Yaskawa INFORM job: SKRZYNIA_4840_0_STOPNI_2OBR.JBI

/JOB
//NAME SKRZYNIA_4840_0_STOPNI_2OBR
///FOLDERNAME 02-SKRZYNIE_JOBS
//POS
///NPOS 694,694,0,51,0,0
///TOOL 0
///POSTYPE PULSE
///PULSE
C00000=1055,-24125,84372,288,19725,204
C00001=0,-15438,65714,0,-68532,0
C00002=4718,-16587,59952,3396,-65485,-935
C00003=32997,-21499,42555,27623,-61436,21376
C00004=31759,-20688,42932,26837,-60850,21559
C00005=28987,-21156,42712,24818,-60442,22222
C00006=33447,-21964,42352,27886,-61721,21330
C00007=37687,-23357,41794,30651,-63289,20620
C00008=38979,-19018,48057,32961,-64962,20678
C00009=37261,-18075,48526,31902,-64209,20901
C00010=35830,-17198,48994,31015,-63571,21092
C00011=34080,-17614,48768,29780,-63290,21485
C00012=37261,-18075,48526,31902,-64209,20901
C00013=4718,-16587,59952,3396,-65485,-935
C00014=32997,-21499,42555,27623,-61436,21376
C00015=31759,-20688,42932,26837,-60850,21559
C00016=28987,-21156,42712,24818,-60442,22222
C00017=33447,-21964,42352,27886,-61721,21330
C00018=37687,-23357,41794,30651,-63289,20620
C00019=38979,-19018,48057,32961,-64962,20678
C00020=37261,-18075,48526,31902,-64209,20901
C00021=35830,-17198,48994,31015,-63571,21092
C00022=34080,-17614,48768,29780,-63290,21485
C00023=37261,-18075,48526,31902,-64209,20901
C00024=47373,-21912,40596,41149,-66086,26950
C00025=45033,-20851,41104,39798,-65001,27223
C00026=42790,-19693,41704,38494,-63946,27495
C00027=41070,-20182,41442,37324,-63566,27891
C00028=45033,-20851,41104,39798,-65001,27223
C00029=45033,-20851,41104,39798,-65001,27223
C00030=59624,-29540,14278,64846,-60867,16042
C00031=57357,-28542,14780,63940,-59509,16120
C00032=56188,-29140,14476,63237,-58995,16387
C00033=59588,-29370,14363,64862,-60819,16012
C00034=54896,-47461,-5979,49852,-59285,4360
C00035=10104,-46603,4759,11228,-37390,-5046
C00036=0,-52280,40443,0,6876,0
C00037=1529,-42140,58025,-5964,2417,3265
C00038=0,-38374,23626,-1605,-51738,268
C00039=63773,-21017,30186,64198,-68685,10387
C00040=61397,-24232,22270,64115,-66256,9272
C00041=59945,-23569,22659,63511,-65413,9334
C00042=58737,-24250,22260,62835,-64893,9588
C00043=61397,-24232,22270,64115,-66256,9272
C00044=45044,-23015,37260,35797,-71879,25522
C00045=39973,-29571,18873,35060,-63052,24165
C00046=38620,-28701,19269,34339,-62304,24363
C00047=36409,-29254,19014,32896,-61805,24958
C00048=44451,-29039,21934,37281,-65892,23702
C00049=49472,-39353,6917,53118,-50908,20251
C00050=45058,-39356,3832,51653,-47640,20099
C00051=42883,-38319,4163,50577,-46309,20295
C00052=40255,-38926,3967,48502,-45334,21060
C00053=46774,-39679,3737,52663,-48537,19827
C00054=48708,-40455,3517,53615,-49689,19657
C00055=43798,-39237,3871,50850,-47027,20335
C00056=41951,-38324,4161,49930,-45891,20507
C00057=39836,-38844,3994,48234,-45126,21137
C00058=48489,-40338,3551,53521,-49551,19665
C00059=1148,-56354,34370,-23,3827,-9
C00060=1148,-56354,34370,-23,3827,-9
C00061=48489,-40338,3551,53521,-49551,19665
C00062=44432,-39026,3936,51363,-47247,20139
C00063=42487,-38069,4248,50403,-46050,20315
C00064=39061,-38795,4009,47695,-44769,21310
C00065=44432,-39026,3936,51363,-47247,20139
C00066=43521,-36748,12770,50182,-45701,23408
C00067=41846,-35383,13175,49516,-44517,23399
C00068=39971,-34448,13485,48491,-43408,23582
C00069=37453,-34980,13306,46330,-42542,24334
C00070=41846,-35383,13175,49516,-44517,23399
C00071=78369,-41260,16071,67181,-65880,21417
C00072=137,-45861,52341,97,-67596,-14
C00073=-31499,-58302,-23356,15027,12889,-13082
C00074=-52768,-43016,-26078,18373,38595,-18774
C00075=-89470,-32103,-32973,29905,69139,-31512
C00076=-68838,-26884,-24872,16972,64732,-23076
C00077=-53036,-11528,-12218,12363,64665,-17409
C00078=-51536,-9474,-10276,11905,64649,-16876
C00079=-51739,-9114,-7787,12104,63269,-17104
C00080=-53036,-11528,-12218,12363,64665,-17409
C00081=-17541,-26226,-24397,927,59032,-5038
C00082=-17541,-26226,-24397,927,59032,-5038
C00083=-16950,-23991,-22741,715,59568,-4818
C00084=-17036,-23563,-20101,755,58071,-4857
C00085=-17541,-26226,-24397,927,59032,-5038
C00086=34102,-23192,-21614,-15638,64271,13209
C00087=33423,-21885,-20599,-15423,64418,12942
C00088=32426,-19856,-18975,-15106,64629,12551
C00089=32578,-19611,-17013,-15290,63535,12762
C00090=33423,-21885,-20599,-15423,64418,12942
C00091=59339,-6070,-6417,-20979,72191,20891
C00092=59339,-6070,-6417,-20979,72191,20891
C00093=57897,-4256,-4562,-20702,71913,20431
C00094=58108,-3992,-2506,-20878,70835,20713
C00095=59339,-6070,-6417,-20979,72191,20891
C00096=42744,-35904,-30225,-18322,62562,16651
C00097=-53036,-11528,-12218,12363,64665,-17409
C00098=-77982,-26538,-29134,27151,66629,-27745
C00099=-70983,-8594,-1966,26503,59809,-49670
C00100=-80152,19776,40785,37351,72704,-50428
C00101=-79984,20154,42529,37516,71911,-50638
C00102=-79233,18397,40079,37458,71885,-50340
C00103=-79984,20154,42529,37516,71911,-50638
C00104=-73519,23289,38838,28890,77081,-45618
C00105=-73519,24511,42682,29072,75582,-46027
C00106=-73519,23289,38838,28890,77081,-45618
C00107=-88897,15706,42282,50101,71325,-56974
C00108=-88897,15706,42282,50101,71325,-56974
C00109=-87612,12343,37838,50071,70996,-56519
C00110=-85283,14202,40272,50301,69633,-56165
C00111=-87338,12550,38107,50098,70839,-56476
C00112=-84952,-1789,13569,34660,47724,-58955
C00113=-67641,-1674,11109,10330,44856,-44725
C00114=-66443,961,13975,9688,44721,-44210
C00115=-67641,-1674,11109,10330,44856,-44725
C00116=-67641,-376,15347,10694,42950,-44967
C00117=-67641,-1674,11109,10330,44856,-44725
C00118=-79040,417,20398,15965,28992,-57786
C00119=-76655,5212,30978,15501,25024,-57306
C00120=-76655,6949,35816,16758,23084,-57955
C00121=-76655,5212,30978,15501,25024,-57306
C00122=-74761,6919,33010,13466,24593,-56049
C00123=-80460,-2874,12270,15804,32253,-57809
C00124=-61258,-29124,-13156,26560,43617,-22150
C00125=-30420,-40507,-29240,27153,53235,15188
C00126=-18589,-38725,-21450,23338,47896,18931
C00127=-17722,-35233,-16455,23322,46926,19051
C00128=-17722,-33749,-12435,23948,45421,18620
C00129=-17722,-33892,-12819,23887,45564,18661
C00130=-16677,-31133,-11209,23138,46167,19311
C00131=-17819,-35820,-17540,23246,47228,19090
C00132=-74104,-11494,-6266,31916,75042,4269
C00133=-71226,-7329,2631,32115,71468,4273
C00134=-71226,-6504,5446,32343,70365,3922
C00135=-71226,-6611,5086,32313,70505,3967
C00136=-68386,-4058,7675,32040,69573,4789
C00137=-73314,-9412,-353,32206,72648,3829
C00138=51751,-31069,-22965,-10739,49070,48663
C00139=49028,-23852,-11575,-9841,46366,47823
C00140=49028,-23004,-8935,-10039,45204,47956
C00141=49028,-23118,-9286,-10013,45357,47939
C00142=47000,-20813,-7527,-8928,45644,47024
C00143=50476,-26208,-15307,-10408,47325,48332
C00144=90602,-5375,6902,-38786,69848,59444
C00145=83174,19950,50269,-44999,67580,58220
C00146=82362,17902,47383,-44926,67511,57879
C00147=83515,19072,48341,-44798,68200,58056
C00148=78091,19382,40247,-36371,72286,52960
C00149=78091,20664,44011,-36670,70997,53443
C00150=78091,19382,40247,-36371,72286,52960
C00151=88699,7296,38566,-55615,63182,60372
C00152=86803,3068,32674,-55410,62638,59657
C00153=84852,4315,34115,-55564,61561,59330
C00154=86803,3068,32674,-55410,62638,59657
C00155=92770,-2803,21719,-53893,67577,59421
C00156=73393,-10627,10934,-27897,30744,62458
C00157=70789,-6606,18800,-27824,27830,62140
C00158=69654,-4593,20814,-26755,27596,61444
C00159=70789,-6606,18800,-27824,27830,62140
C00160=70789,-5070,23059,-29482,26284,63017
C00161=70789,-6606,18800,-27824,27830,62140
C00162=83486,-8736,6503,-27040,35338,66550
C00163=77831,-2041,26192,-25270,18452,68895
C00164=77967,1961,32070,-26860,17569,69698
C00165=77967,5243,40752,-32914,14549,72656
C00166=77967,1961,32070,-26860,17569,69698
C00167=74560,4730,35257,-21622,16551,66717
C00168=77967,1961,32070,-26860,17569,69698
C00169=81109,-22356,2664,-22493,33121,60116
C00170=86168,-49730,-13668,-23926,46819,49343
C00171=44183,-52048,-7537,-24795,46064,51426
C00172=0,-52280,40443,0,6876,0
C00173=0,-52280,40443,0,6876,0
C00174=33629,-57276,-6399,46271,-24969,-2804
C00175=75493,-63502,-64712,103874,-64610,-6298
C00176=47968,-58405,-62693,109749,-46222,-10681
C00177=44214,-60060,-65896,114303,-43519,-9276
C00178=55379,-67378,-68041,108237,-48773,-4935
C00179=62671,-64213,-64640,104431,-56093,-7372
C00180=28458,-50318,6850,47420,-25887,-3347
C00181=0,-52280,40443,0,6876,0
C00182=1055,-24125,84372,288,19725,204
C00183=0,-15438,65714,0,-68532,0
C00184=0,-15438,65714,966,-70097,42926
C00185=69988,-9219,57065,61610,-82752,27767
C00186=63113,-6157,59685,58080,-79692,28271
C00187=46135,-5501,68028,40160,-75108,29748
C00188=49471,-5188,67710,43421,-76082,29577
C00189=63113,-6157,59685,58080,-79692,28271
C00190=69988,-9219,57065,61610,-82752,27767
C00191=0,-15438,65714,966,-70097,42926
C00192=0,-15438,65714,0,-68532,0
C00193=1055,-24125,84372,288,19725,204
C00194=1055,-24125,84372,288,19725,204
C00195=0,-41971,13909,0,6774,1
C00196=-55064,-17017,13106,20113,45767,-35735
C00197=-85641,-3161,12660,31281,67420,-55579
C00198=-77611,9747,38455,32702,57795,-55547
C00199=-77611,9747,38455,32702,57795,-55547
C00200=-80481,23547,61641,37204,60115,-56891
C00201=-80479,11681,28780,33754,71138,-52780
C00202=-73572,15026,34389,33675,67405,-51294
C00203=-73572,20195,49236,35290,62248,-53161
C00204=-82806,26311,53816,38180,73291,-53604
C00205=-71695,3747,16001,30713,64750,-51022
C00206=-70421,5575,20105,30867,63066,-51036
C00207=-35543,-20105,-5144,22821,50284,-40173
C00208=-37830,-23193,-8618,23571,50957,-40982
C00209=11136,-28839,-12562,1025,41780,-20887
C00210=20486,-27077,-7346,-12554,38415,-10736
C00211=59545,-9921,5571,-27063,51925,3267
C00212=55110,-17412,-5825,-19778,50988,-2825
C00213=79390,11759,28162,-35512,71262,52960
C00214=74811,13878,33986,-35807,67493,52464
C00215=74942,18762,48004,-37392,62815,54352
C00216=76815,18630,46530,-37158,64288,54543
C00217=79390,11759,28162,-35512,71262,52960
C00218=10831,-54278,-29128,-6468,39852,-5090
C00219=-67200,-10549,24402,-3189,24913,-39001
C00220=-75122,-2194,12822,3152,39225,-43427
C00221=-77516,10189,32861,8493,33365,-45533
C00222=-75154,17575,49272,7885,27457,-44928
C00223=-68113,9932,38901,1157,28472,-40453
C00224=-67114,5383,31515,9208,32648,-43213
C00225=-66450,3998,29285,10896,33890,-43630
C00226=-66374,3101,28136,14657,35566,-44954
C00227=-66576,452,24763,27028,43375,-49112
C00228=-69928,4230,30673,35488,50431,-52676
C00229=-77050,-3138,8526,33226,61087,-51698
C00230=-67200,-10549,24402,-3189,24913,-39001
C00231=0,-52280,40443,83103,28146,-16510
C00232=99993,-20782,22705,-13349,24734,56519
C00233=67200,-10549,24402,3189,24913,39001
C00234=75122,-2194,12822,-3152,39225,43427
C00235=74323,5203,27259,-5972,33194,43789
C00236=74015,16414,48063,-6821,27325,44224
C00237=56519,1138,28747,9235,29393,33453
C00238=55467,619,28251,10155,29461,32830
C00239=56374,-724,25854,4078,30541,35419
C00240=56480,-7201,15910,-17697,38451,43334
C00241=68252,956,25699,-34035,49810,51639
C00242=77050,-3138,8526,-33226,61087,51698
C00243=67200,-10549,24402,3189,24913,39001
C00244=0,-52280,40443,-83103,28146,16510
C00245=-99993,-20782,22705,13349,24734,-56519
C00246=-91125,453,39555,30378,52425,-51131
C00247=-81425,-5449,14825,37552,56592,-47667
C00248=-81425,-10835,-2515,34915,62871,-45127
C00249=-79239,4305,16082,37593,68846,-50182
C00250=-81302,5892,27588,46359,62943,-54679
C00251=-82227,19402,59913,51524,57300,-60581
C00252=-84844,8890,27031,38640,69740,-53449
C00253=-90096,4679,14083,37467,76581,-51973
C00254=-87885,29238,52923,40761,81198,69685
C00255=-84355,23847,39024,40698,83720,72224
C00256=-81960,27335,46957,41070,80536,71891
C00257=-82643,24718,50492,48951,72637,70260
C00258=-90480,18737,31939,47254,81986,71631
C00259=-94217,10634,17426,46901,86469,-59967
C00260=-81425,-10835,-2515,34915,62871,-45127
C00261=-81425,-5449,14825,37552,56592,-47667
C00262=-94290,-610,44819,32366,49686,-53459
C00263=0,-55136,17047,60468,32096,-4233
C00264=99993,-20782,22705,-13349,24734,56519
C00265=91125,453,39555,-30378,52425,51131
C00266=81425,-5449,14825,-37552,56592,47667
C00267=81425,-10835,-2515,-34915,62871,45127
C00268=79239,4305,16082,-37593,68846,50182
C00269=83239,4964,30263,-50637,62037,57149
C00270=83991,16425,61235,-57769,55250,63273
C00271=93928,7973,40920,-53095,64494,61640
C00272=75109,22299,39152,-26915,78743,47998
C00273=79256,17348,34699,-33448,76412,88212
C00274=79932,23608,50901,-39863,71219,88955
C00275=76220,30771,63034,-41386,67395,88927
C00276=86322,16060,37848,-39554,76452,89287
C00277=87424,-1569,9538,-38190,72401,52253
C00278=81425,-10835,-2515,-34915,62871,45127
C00279=92850,-11266,9233,-39092,60986,50964
C00280=28366,-40369,19479,-5635,23506,17663
C00281=-80334,-19501,31260,21216,42469,-40219
C00282=-80621,-32280,-9061,25825,59412,-41877
C00283=-80621,-37319,-22868,24573,64555,-40576
C00284=-75108,-2453,16462,35304,60348,-42510
C00285=-72231,7240,33473,36511,55681,-43130
C00286=-35770,-19109,7486,28512,40799,-31761
C00287=-39606,-22901,-1163,28356,44724,-32188
C00288=15344,-29112,-5358,-2858,33820,-6852
C00289=13390,-24012,2637,-1527,32105,-7853
C00290=57983,-8601,15571,-27088,42703,12849
C00291=60973,-17187,4937,-27817,44388,13718
C00292=60973,-17187,4937,-27817,44388,13718
C00293=-13287,-42463,-12044,19170,31021,-23010
C00294=-17374,-21287,20534,22794,29118,-26096
C00295=13276,-20759,18622,-1911,29377,-7028
C00296=39924,-14247,19329,-14795,35999,4396
C00297=41528,-14133,18797,-15449,36702,5040
C00298=57001,-5890,26499,-21893,40771,11494
C00299=64054,-19541,3059,-29141,44956,15011
C00300=51466,-33957,-1499,-46586,51805,23434
C00301=17032,-20770,22044,-28854,30468,11088
C00302=-9868,-18638,14971,-8492,38486,-5199
C00303=-40562,-13194,19800,9508,35447,-20184
C00304=-41848,-12620,20103,10165,35810,-20773
C00305=-57278,-4046,28217,17578,39066,-27653
C00306=-71680,-19835,10874,33863,39440,-36917
C00307=-20806,-37586,-12792,9951,42782,-18031
C00308=29087,-45372,27330,-13325,19529,9021
C00309=0,-52280,40443,0,6876,0
C00310=0,-52280,40443,0,6876,0
C00311=0,-52280,40443,0,6876,0
C00312=0,-52280,40443,0,-40718,0
C00313=32359,-35955,27464,28918,-49457,29587
C00314=33244,-30989,28192,31082,-46894,28340
C00315=21151,-27492,32720,20239,-44670,31873
C00316=21536,-57229,-33277,36819,-24396,22621
C00317=20406,-52755,-25486,23563,-35235,28276
C00318=29904,-46498,-2819,27004,-47536,28031
C00319=45803,-31685,22885,64496,-39050,18987
C00320=0,-52277,40442,0,6872,2
C00321=0,-38538,66749,0,-898,0
C00322=0,-52280,40443,0,-79033,35417
C00323=46775,-35113,22190,42926,-67531,20697
C00324=52587,-26056,25345,47610,-66542,17970
C00325=45775,-25572,24450,44032,-63158,18875
C00326=45891,-27794,19511,44698,-62000,18216
C00327=53914,-29436,22058,48262,-67266,17843
C00328=63113,-6157,59685,58080,-79692,28271
C00329=47789,-6280,67353,41142,-75661,29541
C00330=47201,-5612,67930,40804,-75418,29594
C00331=49592,-5172,67757,43430,-76113,29541
C00332=58547,-7653,65645,48613,-79176,28479
C00333=46775,-35113,22190,42926,-67531,20697
C00334=0,-52280,40443,0,-79033,35417
C00335=0,-38922,70509,0,-71891,28081
C00336=0,-38922,70509,0,-71891,28081
C00337=36958,-10079,72709,30464,-66560,20948
C00338=30513,-4130,80544,25739,-66271,22156
C00339=4090,-36983,1084,-1138,-53633,29170
C00340=13946,-45192,10090,9828,-39459,25958
C00341=404,-42897,57020,-1574,2523,869
C00342=0,-52280,40443,0,6876,0
C00343=-99253,-13690,44082,59847,13407,-31313
C00344=-87814,-12734,20141,45739,-14352,-64418
C00345=-86669,-6582,30812,41148,-16781,-62025
C00346=-85055,-5827,31548,44003,-17420,-63187
C00347=-85971,-6262,31124,42409,-17052,-62539
C00348=-86650,-5303,32069,41395,-16716,-62141
C00349=-94954,-14494,-1860,-7818,15857,-59130
C00350=-94509,1544,30797,-849,15127,-60471
C00351=-94509,4151,37772,-1041,12286,-60378
C00352=-88011,-10036,27574,37950,-16527,-60658
C00353=-86125,-12470,22545,29004,-25567,-58412
C00354=-85732,-21202,11427,30682,-24763,-59235
C00355=-84150,-10929,23786,31981,-25941,-59678
C00356=-83036,-10419,24246,33504,-26268,-60308
C00357=-84150,-10929,23786,31981,-25941,-59678
C00358=-85291,-9507,25078,30650,-25411,-59154
C00359=-84150,-10929,23786,31981,-25941,-59678
C00360=-85786,-16909,14677,31743,-23900,-59790
C00361=-84150,-10498,24888,31517,-26306,-59436
C00362=-83174,-10052,25293,32841,-26587,-59984
C00363=-84150,-10498,24888,31517,-26306,-59436
C00364=-85258,-9112,26156,30226,-25800,-58928
C00365=-84150,-10498,24888,31517,-26306,-59436
C00366=-87841,-18519,13420,28367,-23534,-58339
C00367=-84150,-10465,24972,31484,-26336,-59417
C00368=-83241,-10052,25348,32714,-26598,-59924
C00369=-84150,-10465,24972,31484,-26336,-59417
C00370=-85145,-9228,26102,30329,-25881,-58963
C00371=-84150,-10465,24972,31484,-26336,-59417
C00372=-86371,-18277,13606,30568,-23951,-59265
C00373=-84345,-11688,21985,32461,-25312,-59957
C00374=-83211,-11173,22442,34044,-25650,-60618
C00375=-84345,-11688,21985,32461,-25312,-59957
C00376=-85283,-10526,23025,31366,-24861,-59525
C00377=-84345,-11688,21985,32461,-25312,-59957
C00378=-86191,-19647,12567,30467,-24278,-59187
C00379=-84345,-10877,24073,31552,-26006,-59481
C00380=-83051,-10286,24607,33321,-26381,-60213
C00381=-84345,-10877,24073,31552,-26006,-59481
C00382=-85179,-9842,25009,30582,-25619,-59100
C00383=-84345,-10877,24073,31552,-26006,-59481
C00384=-85438,-18022,14839,31140,-24818,-59429
C00385=-84247,-11820,22550,32049,-25753,-59727
C00386=-84104,-10976,23642,32111,-25899,-59738
C00387=-82990,-10465,24105,33639,-26227,-60372
C00388=-84104,-10976,23642,32111,-25899,-59738
C00389=-84898,-9998,24525,31196,-25529,-59378
C00390=-84104,-10976,23642,32111,-25899,-59738
C00391=-86610,-16845,14732,30573,-23614,-59301
C00392=-84104,-10864,23927,31990,-25993,-59674
C00393=-82824,-10273,24459,33737,-26370,-60397
C00394=-84104,-10864,23927,31990,-25993,-59674
C00395=-84789,-10021,24690,31200,-25673,-59363
C00396=-84104,-10864,23927,31990,-25993,-59674
C00397=-83806,-19585,12613,33764,-25080,-60559
C00398=-83924,-10205,25475,31619,-26533,-59453
C00399=-82780,-9675,25960,33156,-26866,-60087
C00400=-83924,-10205,25475,31619,-26533,-59453
C00401=-84478,-9530,26093,30986,-26280,-59206
C00402=-83924,-10205,25475,31619,-26533,-59453
C00403=-87149,-17993,13826,29513,-23647,-58830
C00404=-84920,-13182,20975,31162,-25481,-59361
C00405=-83711,-10572,24852,32056,-26475,-59649
C00406=-82779,-10142,25241,33309,-26748,-60166
C00407=-83711,-10572,24852,32056,-26475,-59649
C00408=-84370,-9774,25579,31305,-26170,-59356
C00409=-83711,-10572,24852,32056,-26475,-59649
C00410=-83642,-3679,42021,23358,-36761,-56118
C00411=-85886,-5975,41264,18964,-40261,-54782
C00412=-83919,-11632,22322,32811,-25616,-60079
C00413=-82884,-11162,22742,34234,-25925,-60671
C00414=-83919,-11632,22322,32811,-25616,-60079
C00415=-84723,-10654,23196,31887,-25230,-59715
C00416=-83919,-11632,22322,32811,-25616,-60079
C00417=-87348,-16035,7353,17528,-35245,-56477
C00418=-86244,-15062,8172,18754,-35315,-57058
C00419=-86244,-16649,3638,19674,-33501,-57585
C00420=-85308,-16228,3988,20718,-33648,-58082
C00421=-86244,-16649,3638,19674,-33501,-57585
C00422=-86740,-15973,4201,19194,-33277,-57362
C00423=-86244,-16649,3638,19674,-33501,-57585
C00424=-73780,-8639,20128,34258,-51705,-52097
C00425=-90711,-17528,-28778,11328,-28245,-57111
C00426=-92565,-19610,-33223,7138,-24591,-57051
C00427=-91512,-19116,-32812,8551,-24603,-57834
C00428=-92565,-19610,-33223,7138,-24591,-57051
C00429=-93003,-18716,-32476,6600,-24397,-56752
C00430=-92565,-19610,-33223,7138,-24591,-57051
C00431=-92565,-19610,-33223,7138,-24591,-57051
C00432=-95836,-54375,-51122,6031,-17685,-48210
C00433=-95836,-54375,-51122,6031,-17685,-48210
C00434=-43821,-47238,-2775,-3022,56549,-3681
C00435=-20126,-26882,59542,2406,16879,-9162
C00436=-20126,-26882,59542,2406,16879,-9162
C00437=98601,-10520,92678,4674,-40855,-9615
C00438=95537,-19831,-2695,-2933,-44471,35837
C00439=92548,-20391,-28429,-6186,-30623,55200
C00440=91429,-17018,-28974,-8057,-27827,56250
C00441=91429,-17018,-28974,-8057,-27827,56250
C00442=90371,-16495,-28521,-9286,-27856,56953
C00443=91429,-17018,-28974,-8057,-27827,56250
C00444=92033,-15799,-27911,-7415,-27588,55880
C00445=91429,-17018,-28974,-8057,-27827,56250
C00446=92548,-20391,-28429,-6186,-30623,55200
C00447=91156,-15018,-4648,-8036,-38181,54813
C00448=90585,-14766,-4428,-8565,-38201,55100
C00449=88830,-13959,-3717,-10186,-38284,55977
C00450=89897,-14456,-4157,-9202,-38230,55445
C00451=90761,-12944,-2809,-8452,-37927,55043
C00452=89897,-14456,-4157,-9202,-38230,55445
C00453=89670,-8466,73559,-9449,-60959,55261
C00454=89910,-11217,67535,-9455,-58896,55399
C00455=85786,-16735,14816,-31782,-23869,59812
C00456=83514,-12996,17929,-35760,-24132,61552
C00457=82251,-12406,18443,-37550,-24551,62308
C00458=83514,-12996,17929,-35760,-24132,61552
C00459=84258,-12095,18717,-34917,-23742,61217
C00460=83514,-12996,17929,-35760,-24132,61552
C00461=87149,-17993,13826,-29513,-23647,58830
C00462=83118,-12818,18089,-36330,-24263,61791
C00463=81915,-12248,18589,-38020,-24666,62504
C00464=83118,-12818,18089,-36330,-24263,61791
C00465=83897,-11882,18912,-35460,-23856,61445
C00466=83118,-12818,18089,-36330,-24263,61791
C00467=83806,-19585,12613,-33764,-25080,60559
C00468=82998,-13006,17925,-36445,-24332,61826
C00469=81675,-12378,18472,-38297,-24777,62607
C00470=82998,-13006,17925,-36445,-24332,61826
C00471=83876,-11958,18841,-35466,-23874,61442
C00472=82998,-13006,17925,-36445,-24332,61826
C00473=86610,-16845,14732,-30573,-23614,59301
C00474=82493,-13239,17725,-37070,-24559,62089
C00475=81406,-12724,18174,-38578,-24928,62723
C00476=82493,-13239,17725,-37070,-24559,62089
C00477=83436,-12134,18690,-36041,-24064,61684
C00478=82493,-13239,17725,-37070,-24559,62089
C00479=84814,-16043,15376,-33312,-24093,60464
C00480=82555,-13613,17404,-36910,-24580,62015
C00481=81384,-13062,17878,-38534,-24974,62698
C00482=82555,-13613,17404,-36910,-24580,62015
C00483=83566,-12434,18427,-35805,-24047,61580
C00484=82555,-13613,17404,-36910,-24580,62015
C00485=86191,-19647,12567,-30467,-24278,59187
C00486=82500,-13648,17375,-36975,-24607,62039
C00487=81467,-13161,17792,-38413,-24955,62645
C00488=82500,-13648,17375,-36975,-24607,62039
C00489=83481,-12505,18364,-35905,-24087,61617
C00490=82500,-13648,17375,-36975,-24607,62039
C00491=86371,-18277,13606,-30568,-23951,59265
C00492=82904,-13790,17251,-36416,-24470,61808
C00493=81715,-13237,17726,-38081,-24865,62509
C00494=82904,-13790,17251,-36416,-24470,61808
C00495=83686,-12878,18037,-35556,-24055,61469
C00496=82904,-13790,17251,-36416,-24470,61808
C00497=87841,-18519,13420,-28367,-23534,58339
C00498=82748,-13879,17174,-36603,-24542,61883
C00499=81692,-13388,17594,-38077,-24893,62505
C00500=82748,-13879,17174,-36603,-24542,61883
C00501=83607,-12881,18032,-35663,-24082,61515
C00502=82748,-13879,17174,-36603,-24542,61883
C00503=85786,-16909,14677,-31743,-23900,59790
C00504=82520,-14198,16902,-36833,-24674,61972
C00505=81460,-13708,17319,-38301,-25026,62591
C00506=82520,-14198,16902,-36833,-24674,61972
C00507=83571,-12989,17938,-35691,-24113,61524
C00508=82520,-14198,16902,-36833,-24674,61972
C00509=85732,-21202,11427,-30682,-24763,59235
C00510=82398,-14365,16763,-36952,-24745,62014
C00511=81172,-13798,17245,-38643,-25153,62725
C00512=82398,-14365,16763,-36952,-24745,62014
C00513=83600,-12984,17944,-35650,-24102,61504
C00514=82398,-14365,16763,-36952,-24745,62014
C00515=86140,-12802,12665,-93523,-10743,85795
C00516=86140,-12802,12665,-93523,-10743,85795
C00517=85030,-12289,13120,-93723,-11463,85776
C00518=86140,-12802,12665,-93523,-10743,85795
C00519=86958,-11660,13681,-94506,-10238,86349
C00520=85239,-16743,-4327,42764,21357,45785
C00521=86674,107,23869,25042,24033,51593
C00522=86674,2327,30134,27824,21680,50173
C00523=87715,-15254,10554,-91589,-9692,85040
C00524=85045,-36869,-4353,-28502,-22832,52282
C00525=0,-24029,84339,0,19981,0
C00526=0,-24029,84339,0,19981,0
C00527=3172,-24246,80980,3465,15913,689
C00528=-86563,-26985,13879,10257,-21548,-45530
C00529=-86191,-19647,12567,30467,-24278,-59187
C00530=-83221,-13587,17636,37793,-25116,-62228
C00531=-91978,-13833,14560,12391,-18633,-51524
C00532=-94992,-13830,14285,1276,-18012,-46664
C00533=-84074,-17488,11256,38660,-23649,-62784
C00534=-73679,-33270,1000,44272,-31600,-64253
C00535=-86926,-60758,23267,6576,1160,-9545
C00536=0,-52280,40443,0,6876,0
C00537=82475,-58079,26734,835,4084,4444
C00538=97932,-26840,7691,8784,-23444,42538
C00539=87166,-16607,16322,-25365,-24201,56345
C00540=84699,-11354,21752,-29145,-24735,57949
C00541=84804,-11023,22730,-28561,-25071,57659
C00542=85100,-26994,10417,-24982,-28140,55821
C00543=0,-52280,40443,0,6876,0
C00544=0,-52280,40443,0,6876,0
C00545=-90140,-60305,18108,-2708,1721,-7625
C00546=-95594,-27428,6866,-4663,-19832,-42154
C00547=-98688,-13767,16447,-18366,-10080,-35766
C00548=-98967,-3050,34440,-28957,-8622,-29685
C00549=-100063,5316,51567,-32262,-10006,-27560
C00550=-94586,18541,64268,-6451,10518,-43578
C00551=-95535,2380,25473,239,27557,-47214
C00552=-91259,3120,34463,-5130,22041,-43946
C00553=-95333,12702,45733,36,21375,-47085
C00554=-99268,-13088,27343,-18620,-14105,-35021
///LIMIT ON
C00555=-90140,-60305,18108,-2708,1721,-7625
///LIMIT OFF
C00556=0,-52280,40443,0,6876,0
C00557=84259,-57935,27522,-3761,3673,6310
C00558=86507,-39672,4297,-27618,-16640,46340
C00559=73669,-37119,-20783,-92053,-19719,85232
C00560=86539,-20830,1725,-71850,-11773,76853
C00561=90325,-18913,6238,-62161,-7452,70888
C00562=97679,-11879,12650,-55334,4229,66281
C00563=98389,-8856,11720,-15676,14634,48538
C00564=96255,-748,20886,-3277,24061,38276
C00565=95132,-6008,10010,1655,28777,36730
C00566=94050,-4188,7205,-2481,41508,36662
C00567=98126,4908,16834,-5042,41918,38535
C00568=100487,-9453,-1206,-10413,41328,41147
C00569=96250,-19428,-8283,-4838,27297,37910
C00570=86507,-39672,4297,-27618,-16640,46340
C00571=84259,-57935,27522,-3761,3673,6310
C00572=0,-52280,40443,0,6876,0
C00573=0,-27933,77061,0,20812,0
C00574=0,-27933,77061,0,20812,0
C00575=0,-52280,40443,0,6876,0
C00576=-91970,-60791,14435,-3343,512,-9412
C00577=-98647,-24138,10005,-11519,-21203,-39749
C00578=-99883,-13980,22886,-11640,-25090,-40341
C00579=-99702,-9154,61728,-1148,-61809,-40243
C00580=-84328,-13042,29707,23458,-33731,-54641
C00581=-83101,-4179,39208,25894,-34785,-55667
C00582=-82881,-4330,38692,26392,-34479,-55866
C00583=-76259,-18287,26646,31659,-38322,-57579
C00584=-89741,-28009,12101,4461,-28076,-46404
C00585=-91970,-60791,14435,-3343,512,-9412
C00586=0,-52280,40443,0,6876,0
C00587=91083,-60784,14823,-9043,-825,15173
C00588=83869,-19403,12921,-33769,-24740,60260
C00589=83869,-19403,12921,-33769,-24740,60260
C00590=83932,-19538,53415,-33663,-71112,60249
C00591=83932,-19538,53415,-33663,-71112,60249
C00592=82480,-12247,21118,-35440,-26416,60009
C00593=82194,-11433,19802,-37650,-25323,61125
C00594=81904,-9374,24711,-35791,-26879,60109
C00595=79790,-20261,14917,-36681,-28829,60258
C00596=76554,-29711,-1870,-46042,-25952,65654
C00597=91083,-60784,14823,-9043,-825,15173
C00598=0,-52280,40443,0,6876,0
C00599=-91526,-60598,16699,7584,176,-13289
C00600=-81382,-25890,9219,35455,-25500,-59095
C00601=-86453,-20958,12525,30076,-22568,-57089
C00602=-86589,-16097,16237,31250,-21582,-57704
C00603=-98933,-11298,20505,-13970,-18736,-37953
C00604=-98281,-10965,21163,-11559,-18548,-39330
C00605=-85424,-18472,14402,34409,-22969,-58895
C00606=-74746,-27148,8488,44263,-29128,-62418
C00607=-81326,-27507,8265,35533,-26282,-59001
C00608=-91415,-60262,16631,7870,-73,-13734
C00609=24,-24029,84339,7,19981,5
C00610=100404,-52373,45687,-1822,14816,-5144
C00611=75939,-26469,7919,-40869,-29645,63133
C00612=81882,-22565,10470,-35355,-26404,61107
C00613=82801,-12246,21732,-34208,-26055,60642
C00614=91824,-10567,23615,-8659,-22197,49820
C00615=96485,-9539,26282,5686,-23135,43736
C00616=77262,-23244,14300,-38922,-31295,61912
C00617=96357,-33562,33410,58602,-23427,10353
C00618=568,-24029,84339,168,19981,112
C00619=-91970,-60791,14435,-3343,512,-9412
C00620=-98991,-22833,11519,-12824,-17638,-36336
C00621=-86376,-13627,18436,38326,-18406,-58533
C00622=-85581,-10814,20279,41280,-18093,-59893
C00623=-85551,-10406,21021,40925,-18257,-59713
C00624=-86274,-24518,9978,34497,-20333,-56613
C00625=-91684,-53777,2301,20525,-9313,-33684
C00626=-67305,-55044,34987,1504,5690,-2468
C00627=0,-52280,40443,0,6876,0
C00628=77036,-56616,31288,-2531,4707,4197
C00629=84359,-28321,8817,-32860,-20485,54199
C00630=81156,-16932,14874,-39538,-26422,62851
C00631=93321,-15690,11640,-5466,-17578,48664
C00632=90862,-14227,15480,-13346,-19623,51954
C00633=77970,-27630,4721,-41834,-28549,63607
C00634=81111,-35571,7141,-33980,-21909,52006
C00635=82626,-57814,28323,-4146,3364,6346
C00636=0,-52280,40443,0,6876,0
C00637=0,-28135,76691,0,20839,0
C00638=0,-28135,76691,0,20839,0
C00639=-45332,-39712,59352,-1730,18713,2903
C00640=-94065,-8316,59352,-1730,-37754,-40387
C00641=-100331,-14895,33931,-8215,-36518,-40227
C00642=-98931,-8578,39429,-6260,-48307,-43744
C00643=-100336,-4176,46216,-7600,-55875,-44633
C00644=-93952,8947,73671,995,-68520,-43850
C00645=-98791,-3170,32594,-4861,-60761,-43748
C00646=-98723,4324,37855,-4919,-58743,-43677
C00647=-98691,-12730,-17828,-7584,-33364,-41886
C00648=-98599,-14408,-28132,-8909,-27584,-41168
C00649=-99605,-15546,-21493,-8548,-33053,-41326
C00650=-98632,914,40428,-4141,-58435,-42510
C00651=-93952,8947,73671,995,-68520,-43850
C00652=-88754,54,62805,4404,-67858,-45120
C00653=-100222,-4532,45667,-7492,-55263,-44561
C00654=-100331,-14895,33931,-8215,-36518,-40227
C00655=-94065,-8316,59352,-1730,-37754,-40387
C00656=-45544,-32973,71870,-2133,15168,3033
C00657=0,-28135,76691,0,20839,0
C00658=54178,-17846,77779,596,-29686,20997
C00659=54178,-17846,77779,-13502,-29686,20997
C00660=99462,-18987,75418,611,-28919,20989
C00661=98707,-9390,78674,1080,-71212,38250
C00662=98768,-5182,41096,1808,-44974,38308
C00663=100431,1771,51615,3823,-56746,39115
C00664=97953,-6621,17555,2289,-50176,39420
C00665=95834,-5353,18817,760,-50052,40242
C00666=86579,-3733,19265,-13263,-48799,44764
C00667=89140,-11519,-8899,-11291,-36869,46482
C00668=89026,-14065,-21014,-13447,-30614,47708
C00669=90457,-16080,-12990,-9972,-37305,45724
C00670=97953,-6621,17555,2289,-50176,39420
C00671=100431,1771,51615,3823,-56746,39115
C00672=98768,-5182,41096,1808,-44974,38308
C00673=98707,-9390,78674,1080,-71212,38250
C00674=0,-28135,76691,0,20839,0
C00675=0,-28135,76691,0,20839,0
C00676=-91526,-60598,16699,7584,176,-13289
C00677=-81382,-25890,9219,35455,-25500,-59095
C00678=-81382,-25890,9219,35455,-25500,-59095
C00679=-85509,-13950,19358,32213,-22393,-58041
C00680=-96341,-12327,18855,-5124,-17594,-42111
C00681=-97523,-9822,24708,-8570,-19966,-40659
C00682=-84656,-25369,12054,31249,-26195,-57129
C00683=-82652,-57346,29982,2770,3944,-5064
C00684=0,-52280,40443,0,6876,0
C00685=60653,-54633,35892,-1212,5841,2035
C00686=77942,-28227,6869,-38010,-29303,61907
C00687=82500,-13648,17375,-36975,-24607,62039
C00688=80731,-11587,18684,-41654,-25449,63953
C00689=80409,-10373,22284,-40214,-26848,63104
C00690=64389,-31987,5108,-50419,-37074,66126
C00691=60653,-54633,35892,-1212,5841,2035
C00692=0,-52280,40443,0,6876,0
C00693=0,-28167,76633,0,20843,0
BC00000=413138
BC00001=413138
BC00002=295997
BC00003=264574
BC00004=264574
BC00005=264574
BC00006=264574
BC00007=233852
BC00008=284288
BC00009=284288
BC00010=284288
BC00011=284288
BC00012=284288
BC00013=388163
BC00014=356740
BC00015=356740
BC00016=356740
BC00017=356740
BC00018=356740
BC00019=407176
BC00020=407176
BC00021=407176
BC00022=407176
BC00023=407176
BC00024=479433
BC00025=479433
BC00026=479433
BC00027=479433
BC00028=479433
BC00029=530237
BC00030=530237
BC00031=530237
BC00032=530237
BC00033=530237
BC00034=541650
BC00035=503930
BC00036=490792
BC00037=671734
BC00038=689202
BC00039=599769
BC00040=599769
BC00041=599769
BC00042=599769
BC00043=599769
BC00044=689202
BC00045=689202
BC00046=689202
BC00047=689202
BC00048=689202
BC00049=726463
BC00050=726463
BC00051=726463
BC00052=726463
BC00053=726463
BC00054=782137
BC00055=782137
BC00056=782137
BC00057=782137
BC00058=782137
BC00059=672533
BC00060=793147
BC00061=859509
BC00062=850421
BC00063=850421
BC00064=850421
BC00065=850421
BC00066=880215
BC00067=880215
BC00068=880215
BC00069=880215
BC00070=880215
BC00071=889613
BC00072=859901
BC00073=927819
BC00074=927819
BC00075=927819
BC00076=943180
BC00077=943180
BC00078=943180
BC00079=943180
BC00080=943180
BC00081=943180
BC00082=943180
BC00083=943180
BC00084=943180
BC00085=943180
BC00086=943180
BC00087=943180
BC00088=943180
BC00089=943180
BC00090=943180
BC00091=943180
BC00092=943180
BC00093=943180
BC00094=943180
BC00095=943180
BC00096=943180
BC00097=943180
BC00098=943180
BC00099=943180
BC00100=943180
BC00101=943182
BC00102=943182
BC00103=943182
BC00104=943182
BC00105=943182
BC00106=943182
BC00107=943182
BC00108=943182
BC00109=943182
BC00110=943182
BC00111=943182
BC00112=943182
BC00113=943182
BC00114=943182
BC00115=943182
BC00116=943182
BC00117=943182
BC00118=943182
BC00119=943182
BC00120=943182
BC00121=943182
BC00122=943182
BC00123=943182
BC00124=943183
BC00125=943184
BC00126=943184
BC00127=943184
BC00128=943184
BC00129=943184
BC00130=943184
BC00131=943184
BC00132=943184
BC00133=943184
BC00134=943184
BC00135=943184
BC00136=943156
BC00137=943170
BC00138=943170
BC00139=943170
BC00140=943170
BC00141=943170
BC00142=943170
BC00143=943170
BC00144=943184
BC00145=943184
BC00146=943184
BC00147=943184
BC00148=943184
BC00149=943184
BC00150=943184
BC00151=943184
BC00152=943184
BC00153=943184
BC00154=943184
BC00155=943184
BC00156=943184
BC00157=943184
BC00158=943184
BC00159=943184
BC00160=943184
BC00161=943184
BC00162=943184
BC00163=943184
BC00164=943184
BC00165=943184
BC00166=943184
BC00167=943184
BC00168=943184
BC00169=911399
BC00170=884954
BC00171=838173
BC00172=801291
BC00173=727925
BC00174=734552
BC00175=750834
BC00176=750837
BC00177=811927
BC00178=811927
BC00179=760768
BC00180=744267
BC00181=689793
BC00182=413138
BC00183=413138
BC00184=413138
BC00185=408626
BC00186=408626
BC00187=408753
BC00188=347392
BC00189=408626
BC00190=408626
BC00191=413138
BC00192=413138
BC00193=413138
BC00194=505502
BC00195=893917
BC00196=915147
BC00197=918406
BC00198=918406
BC00199=918406
BC00200=918406
BC00201=935268
BC00202=935270
BC00203=935270
BC00204=935270
BC00205=935270
BC00206=935270
BC00207=935270
BC00208=935270
BC00209=935270
BC00210=935269
BC00211=935270
BC00212=935271
BC00213=935271
BC00214=935271
BC00215=935271
BC00216=935271
BC00217=935271
BC00218=930781
BC00219=906929
BC00220=936106
BC00221=936109
BC00222=936109
BC00223=936106
BC00224=936107
BC00225=936108
BC00226=936108
BC00227=936109
BC00228=936109
BC00229=936109
BC00230=906929
BC00231=835535
BC00232=835535
BC00233=906929
BC00234=936106
BC00235=936109
BC00236=936109
BC00237=936109
BC00238=936109
BC00239=936114
BC00240=936121
BC00241=936110
BC00242=936109
BC00243=906929
BC00244=835535
BC00245=835535
BC00246=872997
BC00247=918800
BC00248=938197
BC00249=938199
BC00250=938199
BC00251=938199
BC00252=938199
BC00253=938775
BC00254=938199
BC00255=952138
BC00256=952138
BC00257=952138
BC00258=952138
BC00259=952138
BC00260=938197
BC00261=918800
BC00262=872997
BC00263=873283
BC00264=835535
BC00265=872997
BC00266=918800
BC00267=938197
BC00268=938199
BC00269=938199
BC00270=938199
BC00271=938199
BC00272=938199
BC00273=938199
BC00274=938199
BC00275=938199
BC00276=938199
BC00277=938199
BC00278=938197
BC00279=918800
BC00280=849812
BC00281=864290
BC00282=883850
BC00283=922155
BC00284=922155
BC00285=922155
BC00286=922153
BC00287=922155
BC00288=922155
BC00289=922155
BC00290=922153
BC00291=922155
BC00292=914820
BC00293=922155
BC00294=922155
BC00295=922151
BC00296=922153
BC00297=922197
BC00298=922153
BC00299=922155
BC00300=922155
BC00301=922151
BC00302=922153
BC00303=922155
BC00304=922155
BC00305=922155
BC00306=922155
BC00307=918747
BC00308=805523
BC00309=697681
BC00310=697681
BC00311=809313
BC00312=809313
BC00313=883353
BC00314=883353
BC00315=883353
BC00316=883353
BC00317=883353
BC00318=883353
BC00319=845114
BC00320=802643
BC00321=507816
BC00322=507816
BC00323=552804
BC00324=552804
BC00325=551170
BC00326=493239
BC00327=491979
BC00328=285738
BC00329=285865
BC00330=285441
BC00331=256782
BC00332=256782
BC00333=552804
BC00334=507816
BC00335=507816
BC00336=645858
BC00337=645858
BC00338=645858
BC00339=645858
BC00340=645858
BC00341=586783
BC00342=784098
BC00343=815818
BC00344=902189
BC00345=902189
BC00346=902189
BC00347=902189
BC00348=902189
BC00349=902189
BC00350=902189
BC00351=902189
BC00352=902189
BC00353=902189
BC00354=886827
BC00355=895372
BC00356=895372
BC00357=895372
BC00358=895372
BC00359=895372
BC00360=840744
BC00361=840744
BC00362=840744
BC00363=840744
BC00364=840744
BC00365=840744
BC00366=779300
BC00367=771332
BC00368=771332
BC00369=771332
BC00370=771332
BC00371=771332
BC00372=717855
BC00373=717855
BC00374=717855
BC00375=717855
BC00376=717855
BC00377=717855
BC00378=656405
BC00379=649173
BC00380=649173
BC00381=649173
BC00382=649173
BC00383=649173
BC00384=594961
BC00385=594961
BC00386=594961
BC00387=594961
BC00388=594961
BC00389=594961
BC00390=594961
BC00391=533517
BC00392=525229
BC00393=525229
BC00394=525229
BC00395=525229
BC00396=525229
BC00397=472073
BC00398=472073
BC00399=472073
BC00400=472073
BC00401=472073
BC00402=472073
BC00403=410629
BC00404=405662
BC00405=402968
BC00406=402968
BC00407=402968
BC00408=402968
BC00409=402968
BC00410=402968
BC00411=349186
BC00412=349186
BC00413=349186
BC00414=349186
BC00415=349186
BC00416=349186
BC00417=336469
BC00418=336469
BC00419=336469
BC00420=336469
BC00421=336469
BC00422=336469
BC00423=336469
BC00424=367602
BC00425=367601
BC00426=367601
BC00427=367601
BC00428=367601
BC00429=367601
BC00430=367601
BC00431=425303
BC00432=425303
BC00433=514953
BC00434=463119
BC00435=419862
BC00436=451290
BC00437=484962
BC00438=395463
BC00439=369502
BC00440=369502
BC00441=369502
BC00442=369502
BC00443=369502
BC00444=369502
BC00445=369502
BC00446=369502
BC00447=368885
BC00448=368885
BC00449=368885
BC00450=368885
BC00451=368885
BC00452=368885
BC00453=419064
BC00454=366918
BC00455=349186
BC00456=353241
BC00457=353241
BC00458=353241
BC00459=353241
BC00460=353241
BC00461=410629
BC00462=409135
BC00463=409135
BC00464=409135
BC00465=409135
BC00466=409135
BC00467=472073
BC00468=476126
BC00469=476126
BC00470=476126
BC00471=476126
BC00472=476126
BC00473=533517
BC00474=532644
BC00475=532644
BC00476=532644
BC00477=532644
BC00478=532644
BC00479=594961
BC00480=599988
BC00481=599988
BC00482=599988
BC00483=599988
BC00484=599988
BC00485=656405
BC00486=653254
BC00487=653254
BC00488=653254
BC00489=653254
BC00490=653254
BC00491=717855
BC00492=721570
BC00493=721570
BC00494=721570
BC00495=721570
BC00496=721570
BC00497=779300
BC00498=777963
BC00499=777963
BC00500=777963
BC00501=777963
BC00502=777963
BC00503=840744
BC00504=843810
BC00505=843810
BC00506=843810
BC00507=843810
BC00508=843810
BC00509=902188
BC00510=900128
BC00511=900128
BC00512=900128
BC00513=900128
BC00514=900128
BC00515=919406
BC00516=904045
BC00517=904045
BC00518=904045
BC00519=904045
BC00520=904045
BC00521=904045
BC00522=904045
BC00523=904045
BC00524=870060
BC00525=723883
BC00526=723883
BC00527=689791
BC00528=641458
BC00529=721442
BC00530=721442
BC00531=721439
BC00532=781482
BC00533=781888
BC00534=781888
BC00535=781888
BC00536=781888
BC00537=768943
BC00538=718475
BC00539=718475
BC00540=718475
BC00541=778313
BC00542=778313
BC00543=659914
BC00544=792672
BC00545=792672
BC00546=902112
BC00547=902112
BC00548=894618
BC00549=905919
BC00550=888754
BC00551=895231
BC00552=895231
BC00553=895231
BC00554=888755
BC00555=731228
BC00556=746589
BC00557=746589
BC00558=841363
BC00559=910181
BC00560=910181
BC00561=915612
BC00562=910935
BC00563=918536
BC00564=912118
BC00565=911606
BC00566=910354
BC00567=910516
BC00568=894820
BC00569=894820
BC00570=826002
BC00571=792672
BC00572=792672
BC00573=700249
BC00574=546214
BC00575=546214
BC00576=546211
BC00577=546211
BC00578=406776
BC00579=406776
BC00580=352261
BC00581=346119
BC00582=406266
BC00583=406266
BC00584=491556
BC00585=546211
BC00586=546214
BC00587=546214
BC00588=507604
BC00589=410782
BC00590=429690
BC00591=375447
BC00592=350474
BC00593=350474
BC00594=408658
BC00595=408658
BC00596=507604
BC00597=546214
BC00598=546214
BC00599=516757
BC00600=591809
BC00601=591809
BC00602=591809
BC00603=591183
BC00604=650353
BC00605=650538
BC00606=650538
BC00607=584003
BC00608=515801
BC00609=520018
BC00610=520018
BC00611=590597
BC00612=593080
BC00613=593080
BC00614=593080
BC00615=652456
BC00616=652559
BC00617=594788
BC00618=433888
BC00619=546211
BC00620=830322
BC00621=830322
BC00622=830322
BC00623=890247
BC00624=890396
BC00625=798848
BC00626=798848
BC00627=798848
BC00628=798848
BC00629=832296
BC00630=845010
BC00631=845010
BC00632=904605
BC00633=904704
BC00634=818840
BC00635=818839
BC00636=818839
BC00637=526967
BC00638=334612
BC00639=334612
BC00640=334612
BC00641=350464
BC00642=350464
BC00643=359337
BC00644=359337
BC00645=359337
BC00646=359721
BC00647=359453
BC00648=359342
BC00649=359337
BC00650=359337
BC00651=359337
BC00652=359337
BC00653=358620
BC00654=350464
BC00655=334612
BC00656=334612
BC00657=334612
BC00658=334613
BC00659=460273
BC00660=501279
BC00661=334612
BC00662=334610
BC00663=349510
BC00664=365935
BC00665=365935
BC00666=365934
BC00667=348430
BC00668=348430
BC00669=348430
BC00670=365935
BC00671=349510
BC00672=334610
BC00673=334612
BC00674=334612
BC00675=512789
BC00676=516757
BC00677=526627
BC00678=466969
BC00679=466969
BC00680=466969
BC00681=524647
BC00682=525745
BC00683=525745
BC00684=525745
BC00685=525745
BC00686=473911
BC00687=473911
BC00688=473911
BC00689=532824
BC00690=533743
BC00691=525745
BC00692=525745
BC00693=525747
///POSTYPE BASE
///RECTAN
///RCONF 1,0,0,0,0,0,0,0,0,0,0,0,0,0,0,0,0,0,0,0,0,0,0,0
P00006=0.000,0.000,0.000,0.0000,0.0000,0.0000
///RCONF 0,0,0,0,0,0,0,0,0,0,0,0,0,0,0,0,0,0,0,0,0,0,0,0
P00057=0.000,0.000,2.000,0.0000,0.0000,0.0000
P00058=0.000,0.000,3.000,0.0000,0.0000,0.0000
///RCONF 1,0,0,0,0,0,0,0,0,0,0,0,0,0,0,0,0,0,0,0,0,0,0,0
P00097=0.043,-1.896,1.568,0.0000,0.0000,0.0000
P00098=-0.089,-2.467,4.059,0.0000,0.0000,0.0000
P00099=0.011,-2.380,1.226,0.0000,0.0000,0.0000
P00100=-0.081,2.558,4.482,0.0000,0.0000,0.0000
P00101=0.030,-2.286,2.993,0.0000,0.0000,0.0000
P00102=-0.005,-1.108,1.644,0.0000,0.0000,0.0000
P00103=-0.094,-3.400,4.200,0.0000,0.0000,0.0000
P00104=0.043,-2.127,5.826,0.0000,0.0000,0.0000
P00105=-0.043,0.662,5.286,0.0000,0.0000,0.0000
P00106=-0.018,-2.519,0.237,0.0000,0.0000,0.0000
P00107=-0.008,-4.537,-4.500,0.0000,0.0000,0.0000
P00108=0.014,-3.040,2.637,0.0000,0.0000,0.0000
///RCONF 0,0,0,0,0,0,0,0,0,0,0,0,0,0,0,0,0,0,0,0,0,0,0,0
P00299=-1.404,-0.874,9.133,0.0000,0.0000,0.0000
///RCONF 1,0,0,0,0,0,0,0,0,0,0,0,0,0,0,0,0,0,0,0,0,0,0,0
P00301=0.046,-2.112,7.779,0.0000,0.0000,0.0000
P00302=-0.180,-2.409,6.326,0.0000,0.0000,0.0000
///RCONF 0,0,0,0,0,0,0,0,0,0,0,0,0,0,0,0,0,0,0,0,0,0,0,0
P00303=-0.004,-1.437,-4.584,0.0000,0.0000,0.0000
P00304=0.028,-1.666,-4.234,0.0000,0.0000,0.0000
P00305=-0.003,-1.920,-3.501,0.0000,0.0000,0.0000
P00306=0.015,-2.252,-3.054,0.0000,0.0000,0.0000
P00307=0.019,-2.151,-5.077,0.0000,0.0000,0.0000
P00308=-0.003,-2.092,-4.888,0.0000,0.0000,0.0000
P00309=-0.040,-2.205,-4.992,0.0000,0.0000,0.0000
P00310=-0.006,-2.490,-5.925,0.0000,0.0000,0.0000
P00311=-0.007,-2.079,-5.307,0.0000,0.0000,0.0000
P00312=-0.032,2.202,-7.632,0.0000,0.0000,0.0000
///RCONF 1,0,0,0,0,0,0,0,0,0,0,0,0,0,0,0,0,0,0,0,0,0,0,0
P00349=0.060,0.167,-1.133,0.0000,0.0000,0.0000
///RCONF 0,0,0,0,0,0,0,0,0,0,0,0,0,0,0,0,0,0,0,0,0,0,0,0
P00350=11.519,-0.008,1.149,0.0000,0.0000,0.0000
P00351=13.563,-0.027,-0.653,0.0000,0.0000,0.0000
P00352=13.252,-0.027,-0.827,0.0000,0.0000,0.0000
P00353=10.971,-0.082,0.776,0.0000,0.0000,0.0000
P00354=-0.024,2.508,-1.824,0.0000,0.0000,0.0000
P00355=-0.001,2.528,-1.131,0.0000,0.0000,0.0000
P00356=-0.034,2.921,-0.262,0.0000,0.0000,0.0000
P00357=0.003,3.386,-0.091,0.0000,0.0000,0.0000
P00358=0.014,3.037,-0.020,0.0000,0.0000,0.0000
P00359=-0.005,2.731,0.912,0.0000,0.0000,0.0000
P00360=-0.011,3.412,0.438,0.0000,0.0000,0.0000
P00361=0.018,3.050,1.253,0.0000,0.0000,0.0000
P00362=0.014,2.784,0.148,0.0000,0.0000,0.0000
P00399=-2.449,0.031,8.825,0.0000,0.0000,0.0000
P00400=5.920,-3.503,-0.024,0.0000,0.0000,0.0000
P00401=3.430,-0.021,1.131,0.0000,0.0000,0.0000
P00402=-0.253,1.107,3.062,0.0000,0.0000,0.0000
P00403=-3.666,-0.015,5.328,0.0000,0.0000,0.0000
P00405=2.420,0.007,1.427,0.0000,0.0000,0.0000
P00406=3.513,-0.022,0.429,0.0000,0.0000,0.0000
P00415=-1.781,-1.303,3.250,0.0000,0.0000,0.0000
P00416=0.027,1.119,3.078,0.0000,0.0000,0.0000
//INST
///DATE 2025/06/04 08:21
///ATTR SC,RW
///GROUP1 RB1,BS1
NOP
CALL JOB:MOVE_INTO_TUNNEL
SFTOF
'------------------------
'------------------------
'SPOINA SRODEK DOL
'------------------------
'------------------------
MOVJ C00000 BC00000 VJ=10.00
MOVJ C00001 BC00001 VJ=30.00
'------------------------
'PODLOGA_BEZ_ROZPORKI
'------------------------
'TEST
MOVL C00002 BC00002 V=166.7
MOVL C00003 BC00003 V=166.7 PL=0
REFP 3 C00004 BC00004
CALL JOB:SEARCH-R1
IMOV P0057 V=23.0
SET P0097 P0006
SFTON P0097
REFP 3 C00005 BC00005
CALL JOB:SEARCH-R1
SET P0097 P0006
SFTON P0097
MOVL C00006 BC00006 V=166.7 PL=0
SFTOF
COMM MOVL C00007 BC00007 V=333.3
MOVL C00008 BC00008 V=333.3
MOVL C00009 BC00009 V=166.7 PL=0
REFP 3 C00010 BC00010
CALL JOB:SEARCH-R1
IMOV P0057 V=23.0
SET P0098 P0006
SFTON P0098
REFP 3 C00011 BC00011
CALL JOB:SEARCH-R1
SET P0098 P0006
SFTON P0098
MOVL C00012 BC00012 V=166.7 PL=0
'TEST
SFTOF
'------------------------
'W38 P
'------------------------
'TEST
MOVL C00013 BC00013 V=166.7
MOVL C00014 BC00014 V=166.7 PL=0
REFP 3 C00015 BC00015
CALL JOB:SEARCH-R1
IMOV P0057 V=23.0
SET P0099 P0006
SFTON P0099
REFP 3 C00016 BC00016
CALL JOB:SEARCH-R1
SET P0099 P0006
SFTON P0099
MOVL C00017 BC00017 V=166.7 PL=0
'TEST
SFTOF
MOVL C00018 BC00018 V=333.3
MOVL C00019 BC00019 V=333.3
'------------------------
'W38 L
'------------------------
'TEST
MOVL C00020 BC00020 V=166.7 PL=0
REFP 3 C00021 BC00021
CALL JOB:SEARCH-R1
IMOV P0057 V=23.0
SET P0100 P0006
SFTON P0100
REFP 3 C00022 BC00022
CALL JOB:SEARCH-R1
SET P0100 P0006
SFTON P0100
MOVL C00023 BC00023 V=166.7 PL=0
'TEST
SFTOF
MOVJ C00024 BC00024 VJ=20.00
'------------------------
'W45 P
'------------------------
MOVL C00025 BC00025 V=166.7 PL=0
REFP 3 C00026 BC00026
CALL JOB:SEARCH-R1
IMOV P0057 V=23.0
SET P0101 P0006
SFTON P0101
REFP 3 C00027 BC00027
CALL JOB:SEARCH-R1
SET P0101 P0006
SFTON P0101
MOVL C00028 BC00028 V=166.7 PL=0
'TEST
SFTOF
MOVJ C00029 BC00029 VJ=20.00
'------------------------
'W45 L
'------------------------
MOVL C00030 BC00030 V=133.3 PL=0
REFP 3 C00031 BC00031
CALL JOB:SEARCH-R1
IMOV P0057 V=23.0
SET P0102 P0006
SFTON P0102
REFP 3 C00032 BC00032
CALL JOB:SEARCH-R1
SET P0102 P0006
SFTON P0102
MOVL C00033 BC00033 V=250.0 PL=0
'TEST
SFTOF
MOVJ C00034 BC00034 VJ=30.00
MOVJ C00035 BC00035 VJ=30.00
MOVJ C00036 BC00036 VJ=30.00
MOVJ C00037 BC00037 VJ=30.00
MOVJ C00038 BC00038 VJ=20.00
MOVJ C00039 BC00039 VJ=20.00
'------------------------
'W48 P
'------------------------
'TEST
MOVL C00040 BC00040 V=133.3 PL=0
REFP 3 C00041 BC00041
CALL JOB:SEARCH-R1
IMOV P0057 V=23.0
SET P0103 P0006
SFTON P0103
REFP 3 C00042 BC00042
CALL JOB:SEARCH-R1
SET P0103 P0006
SFTON P0103
MOVL C00043 BC00043 V=166.7 PL=0
'TEST
SFTOF
MOVL C00044 BC00044 V=416.7
'------------------------
'W48 L
'------------------------
SFTOF
MOVL C00045 BC00045 V=133.3 PL=0
REFP 3 C00046 BC00046
CALL JOB:SEARCH-R1
IMOV P0057 V=23.0
SET P0104 P0006
SFTON P0104
REFP 3 C00047 BC00047
CALL JOB:SEARCH-R1
SET P0104 P0006
SFTON P0104
MOVL C00048 BC00048 V=166.7 PL=0
SFTOF
MOVJ C00049 BC00049 VJ=20.00
'------------------------
'W36 P
'------------------------
MOVL C00050 BC00050 V=133.3 PL=0
REFP 3 C00051 BC00051
CALL JOB:SEARCH-R1
IMOV P0057 V=23.0
SET P0105 P0006
SFTON P0105
REFP 3 C00052 BC00052
CALL JOB:SEARCH-R1
SET P0105 P0006
SFTON P0105
MOVL C00053 BC00053 V=166.7 PL=0
'TEST
SFTOF
MOVJ C00054 BC00054 VJ=20.00
'------------------------
'W36 L
'------------------------
MOVL C00055 BC00055 V=166.7 PL=0
REFP 3 C00056 BC00056
CALL JOB:SEARCH-R1
IMOV P0057 V=23.0
SET P0106 P0006
SFTON P0106
REFP 3 C00057 BC00057
CALL JOB:SEARCH-R1
SET P0106 P0006
SFTON P0106
SFTOF
MOVL C00058 BC00058 V=166.7 PL=0
MOVJ C00059 BC00059 VJ=25.00
MOVJ C00060 BC00060 VJ=25.00
'TEST
MOVJ C00061 BC00061 VJ=20.00
SFTOF
'------------------------
'W44 P
'------------------------
'TEST
MOVL C00062 BC00062 V=133.3 PL=0
REFP 3 C00063 BC00063
CALL JOB:SEARCH-R1
IMOV P0057 V=23.0
SET P0107 P0006
SFTON P0107
REFP 3 C00064 BC00064
CALL JOB:SEARCH-R1
SET P0107 P0006
SFTON P0107
SFTOF
MOVL C00065 BC00065 V=250.0 PL=0
'TEST
MOVL C00066 BC00066 V=416.7
MOVL C00067 BC00067 V=166.7 PL=0
REFP 3 C00068 BC00068
CALL JOB:SEARCH-R1
IMOV P0057 V=23.0
SET P0108 P0006
SFTON P0108
REFP 3 C00069 BC00069
CALL JOB:SEARCH-R1
SET P0108 P0006
SFTON P0108
SFTOF
MOVL C00070 BC00070 V=250.0 PL=0
'TEST
SFTOF
MOVL C00071 BC00071 V=250.0
MOVJ C00072 BC00072 VJ=25.00
CALL JOB:FRONT_SEARCH_0ST-2_4840_V3
COMM MOVJ C00073 BC00073 VJ=20.00
COMM MOVJ C00074 BC00074 VJ=20.00
COMM MOVJ C00075 BC00075 VJ=20.00
COMM 'DODANE
COMM 'SZUKANIE FRONT
COMM '------------------------
COMM '503
COMM '------------------------
COMM MOVL C00076 BC00076 V=333.3
COMM MOVL C00077 BC00077 V=166.7 PL=0
COMM REFP 3 C00078 BC00078
COMM CALL JOB:SEARCH-R1
COMM IMOV P0058 V=16.7
COMM SET P0350 P0006
COMM SFTON P0350
COMM REFP 3 C00079 BC00079
COMM CALL JOB:SEARCH-R1
COMM SET P0350 P0006
COMM SFTON P0350
COMM MOVL C00080 BC00080 V=66.7 PL=0
COMM SFTOF
COMM '------------------------
COMM '------------------------
COMM '502
COMM '------------------------
COMM MOVL C00081 BC00081 V=166.7
COMM MOVL C00082 BC00082 V=66.7 PL=0
COMM REFP 3 C00083 BC00083
COMM CALL JOB:SEARCH-R1
COMM IMOV P0058 V=16.7
COMM SET P0351 P0006
COMM SFTON P0351
COMM REFP 3 C00084 BC00084
COMM CALL JOB:SEARCH-R1
COMM SET P0351 P0006
COMM SFTON P0351
COMM MOVL C00085 BC00085 V=66.7 PL=0
COMM SFTOF
COMM '------------------------
COMM '------------------------
COMM '501
COMM '------------------------
COMM MOVL C00086 BC00086 V=166.7
COMM MOVL C00087 BC00087 V=66.7 PL=0
COMM REFP 3 C00088 BC00088
COMM CALL JOB:SEARCH-R1
COMM IMOV P0058 V=16.7
COMM SET P0352 P0006
COMM SFTON P0352
COMM REFP 3 C00089 BC00089
COMM CALL JOB:SEARCH-R1
COMM SET P0352 P0006
COMM SFTON P0352
COMM MOVL C00090 BC00090 V=66.7 PL=0
COMM SFTOF
COMM '------------------------
COMM '------------------------
COMM '500
COMM '------------------------
COMM MOVL C00091 BC00091 V=166.7
COMM MOVL C00092 BC00092 V=66.7 PL=0
COMM REFP 3 C00093 BC00093
COMM CALL JOB:SEARCH-R1
COMM IMOV P0058 V=16.7
COMM SET P0353 P0006
COMM SFTON P0353
COMM REFP 3 C00094 BC00094
COMM CALL JOB:SEARCH-R1
COMM SET P0353 P0006
COMM SFTON P0353
COMM MOVL C00095 BC00095 V=66.7 PL=0
COMM SFTOF
COMM '------------------------
COMM MOVL C00096 BC00096 V=333.3
COMM MOVL C00097 BC00097 V=333.3
COMM MOVJ C00098 BC00098 VJ=10.00
COMM 'DODANE
COMM MOVJ C00099 BC00099 VJ=10.00
COMM '------------------------
COMM 'SFT402
COMM '------------------------
COMM SFTOF
COMM MOVL C00100 BC00100 V=150.0
COMM MOVL C00101 BC00101 V=66.7 PL=0
COMM REFP 3 C00102 BC00102
COMM CALL JOB:SEARCH-R1
COMM SET P0402 P0006
COMM SFTON P0402
COMM MOVL C00103 BC00103 V=150.0
COMM MOVL C00104 BC00104 V=66.7 PL=0
COMM REFP 3 C00105 BC00105
COMM CALL JOB:SEARCH-R1
COMM SET P0402 P0006
COMM SFTON P0402
COMM MOVL C00106 BC00106 V=133.3
COMM MOVL C00107 BC00107 V=150.0
COMM MOVL C00108 BC00108 V=150.0
COMM MOVL C00109 BC00109 V=66.7 PL=0
COMM REFP 3 C00110 BC00110
COMM CALL JOB:SEARCH-R1
COMM SET P0402 P0006
COMM SFTOF
COMM MOVL C00111 BC00111 V=150.0
COMM '------------------------
COMM 'SFT403
COMM '------------------------
COMM 'START
COMM SFTOF
COMM MOVL C00112 BC00112 V=250.0
COMM MOVL C00113 BC00113 V=133.3 PL=0
COMM REFP 3 C00114 BC00114
COMM CALL JOB:SEARCH-R1
COMM SET P0416 P0006
COMM SFTON P0416
COMM MOVL C00115 BC00115 V=133.3
COMM REFP 3 C00116 BC00116
COMM CALL JOB:SEARCH-R1
COMM SET P0402 P0006
COMM SFTOF
COMM MOVL C00117 BC00117 V=150.0
COMM '------------------------
COMM '------------------------
COMM SFTOF
COMM MOVL C00118 BC00118 V=250.0
COMM MOVL C00119 BC00119 V=133.3 PL=0
COMM REFP 3 C00120 BC00120
COMM CALL JOB:SEARCH-R1
COMM SET P0403 P0006
COMM SFTON P0403
COMM MOVL C00121 BC00121 V=66.7 PL=0
COMM REFP 3 C00122 BC00122
COMM CALL JOB:SEARCH-R1
COMM SET P0403 P0006
COMM SFTOF
COMM MOVL C00123 BC00123 V=150.0
COMM MOVJ C00124 BC00124 VJ=20.00
COMM MOVJ C00125 BC00125 VJ=20.00
COMM '------------------------
COMM 'SFT401
COMM '------------------------
COMM SFTOF
COMM MOVL C00126 BC00126 V=150.0
COMM MOVL C00127 BC00127 V=66.7 PL=0
COMM REFP 3 C00128 BC00128
COMM CALL JOB:SEARCH-R1
COMM SET P0401 P0006
COMM SFTON P0401
COMM MOVL C00129 BC00129 V=66.7 PL=0
COMM REFP 3 C00130 BC00130
COMM CALL JOB:SEARCH-R1
COMM SET P0401 P0006
COMM SFTOF
COMM MOVL C00131 BC00131 V=150.0
COMM 'SFT400
COMM '------------------------
COMM SFTOF
COMM MOVL C00132 BC00132 V=333.3
COMM MOVL C00133 BC00133 V=66.7 PL=0
COMM REFP 3 C00134 BC00134
COMM CALL JOB:SEARCH-R1
COMM SET P0405 P0006
COMM SFTON P0405
COMM MOVL C00135 BC00135 V=66.7 PL=0
COMM REFP 3 C00136 BC00136
COMM CALL JOB:SEARCH-R1
COMM SET P0405 P0006
COMM SFTOF
COMM MOVL C00137 BC00137 V=150.0
COMM 'SFT400
COMM '------------------------
COMM SFTOF
COMM MOVL C00138 BC00138 V=333.3
COMM MOVL C00139 BC00139 V=133.3 PL=0
COMM REFP 3 C00140 BC00140
COMM CALL JOB:SEARCH-R1
COMM SET P0406 P0006
COMM SFTON P0406
COMM MOVL C00141 BC00141 V=66.7 PL=0
COMM REFP 3 C00142 BC00142
COMM CALL JOB:SEARCH-R1
COMM SET P0406 P0006
COMM SFTOF
COMM MOVL C00143 BC00143 V=150.0
COMM 'SFT400
COMM '------------------------
COMM SFTOF
COMM MOVL C00144 BC00144 V=150.0
COMM MOVL C00145 BC00145 V=66.7 PL=0
COMM REFP 3 C00146 BC00146
COMM CALL JOB:SEARCH-R1
COMM SET P0400 P0006
COMM SFTON P0400
COMM MOVL C00147 BC00147 V=150.0
COMM MOVL C00148 BC00148 V=66.7 PL=0
COMM REFP 3 C00149 BC00149
COMM CALL JOB:SEARCH-R1
COMM SET P0400 P0006
COMM SFTON P0400
COMM MOVL C00150 BC00150 V=150.0
COMM MOVL C00151 BC00151 V=150.0
COMM MOVL C00152 BC00152 V=66.7 PL=0
COMM REFP 3 C00153 BC00153
COMM CALL JOB:SEARCH-R1
COMM SET P0400 P0006
COMM SFTOF
COMM MOVL C00154 BC00154 V=83.3
COMM MOVL C00155 BC00155 V=250.0
COMM MOVL C00156 BC00156 V=333.3
COMM MOVL C00157 BC00157 V=66.7 PL=0
COMM REFP 3 C00158 BC00158
COMM CALL JOB:SEARCH-R1
COMM SET P0415 P0006
COMM SFTON P0415
COMM MOVL C00159 BC00159 V=133.3
COMM REFP 3 C00160 BC00160
COMM CALL JOB:SEARCH-R1
COMM SET P0415 P0006
COMM SFTOF
COMM MOVL C00161 BC00161 V=150.0
COMM '------------------------
COMM 'SFT403
COMM '------------------------
COMM 'START
COMM SFTOF
COMM MOVJ C00162 BC00162 VJ=10.00
COMM '------------------------
COMM 'SFT399
COMM '------------------------
COMM 'START
COMM SFTOF
COMM MOVL C00163 BC00163 V=150.0
COMM MOVL C00164 BC00164 V=66.7 PL=0
COMM REFP 3 C00165 BC00165
COMM CALL JOB:SEARCH-R1
COMM SET P0399 P0006
COMM SFTON P0399
COMM MOVL C00166 BC00166 V=66.7 PL=0
COMM REFP 3 C00167 BC00167
COMM CALL JOB:SEARCH-R1
COMM SET P0399 P0006
COMM SFTOF
COMM MOVL C00168 BC00168 V=150.0
COMM MOVJ C00169 BC00169 VJ=20.00
COMM MOVJ C00170 BC00170 VJ=30.00
MOVJ C00171 BC00171 VJ=30.00
MOVJ C00172 BC00172 VJ=30.00
MOVJ C00173 BC00173 VJ=40.00
'WELD
'WELD
MOVJ C00174 BC00174 VJ=20.00
'**********************
'W36
'**********************
MOVL C00175 BC00175 V=500.0
SFTON P0105
MOVL C00176 BC00176 V=166.7 PL=0
SFTOF
MACRO1 MJ#(0) ARGF24
ARCON
SFTON P0106
MOVL C00177 BC00177 V=11.0
ARCOF
SFTOF
MOVJ C00178 BC00178 VJ=15.00
MOVJ C00179 BC00179 VJ=10.00
MOVJ C00180 BC00180 VJ=10.00
MOVJ C00181 BC00181 VJ=10.00
MOVJ C00182 BC00182 VJ=30.00
MOVJ C00183 BC00183 VJ=20.00
MOVJ C00184 BC00184 VJ=10.00
MOVJ C00185 BC00185 VJ=15.00
'**********************
'W38
'**********************
MOVL C00186 BC00186 V=500.0
SFTON P0100
MOVL C00187 BC00187 V=166.7 PL=0
SFTOF
ARCON
SFTON P0099
MOVL C00188 BC00188 V=11.0
ARCOF
SFTOF
'DODANE
MOVL C00189 BC00189 V=500.0
MOVJ C00190 BC00190 VJ=10.00
MOVJ C00191 BC00191 VJ=10.00
MOVJ C00192 BC00192 VJ=10.00
MOVJ C00193 BC00193 VJ=10.00
MOVJ C00194 BC00194 VJ=25.00
COMM '**********************
COMM '**********************
COMM 'POCZATEK SPAWANIA PRZOD
COMM '**********************
COMM '**********************
COMM MOVJ C00195 BC00195 VJ=30.00
COMM MOVL C00196 BC00196 V=416.7
COMM MOVJ C00197 BC00197 VJ=10.00
COMM MOVJ C00198 BC00198 VJ=10.00
COMM MOVL C00199 BC00199 V=150.0
COMM MOVL C00200 BC00200 V=150.0
COMM '**********************
COMM 'W41A SIDE
COMM '**********************
COMM MOVL C00201 BC00201 V=250.0
COMM SFTON P0402
COMM MOVL C00202 BC00202 V=66.7 PL=0
COMM MACRO1 MJ#(0) ARGF14
COMM ARCON
COMM MOVL C00203 BC00203 V=9.2
COMM ARCOF
COMM SFTOF
COMM MOVL C00204 BC00204 V=166.7
COMM '**********************
COMM 'W41A FRONT
COMM '**********************
COMM MOVL C00205 BC00205 V=250.0
COMM SFTON P0350
COMM MOVL C00206 BC00206 V=66.7 PL=0
COMM SFTOF
COMM MACRO1 MJ#(0) ARGF21
COMM ARCON
COMM SFTON P0351
COMM MOVL C00207 BC00207 V=8.3
COMM SFTOF
COMM ARCOF
COMM MOVL C00208 BC00208 V=166.7
COMM '**********************
COMM 'W41B FRONT
COMM '**********************
COMM MOVL C00209 BC00209 V=250.0
COMM SFTON P0352
COMM MOVL C00210 BC00210 V=66.7 PL=0
COMM SFTOF
COMM MACRO1 MJ#(0) ARGF21
COMM ARCON
COMM SFTON P0353
COMM MOVL C00211 BC00211 V=8.3
COMM SFTOF
COMM ARCOF
COMM MOVL C00212 BC00212 V=166.7
COMM MOVL C00213 BC00213 V=100.0
COMM '**********************
COMM 'W41A SIDE
COMM '**********************
COMM SFTON P0400
COMM MOVL C00214 BC00214 V=66.7 PL=0
COMM MACRO1 MJ#(0) ARGF21
COMM ARCON
COMM MOVL C00215 BC00215 V=8.3
COMM ARCOF
COMM SFTOF
COMM MOVL C00216 BC00216 V=166.7
COMM MOVL C00217 BC00217 V=166.7
COMM MOVL C00218 BC00218 V=333.3
COMM MOVJ C00219 BC00219 VJ=20.00
COMM MOVJ C00220 BC00220 VJ=20.00
COMM '**********************
COMM 'W42A.1
COMM '**********************
COMM 'POPRAWIC
COMM MOVL C00221 BC00221 V=500.0
COMM SFTON P0403
COMM MOVL C00222 BC00222 V=66.7 PL=0
COMM MACRO1 MJ#(0) ARGF9
COMM ARCON
COMM MOVL C00223 BC00223 V=9.2
COMM SFTON P0416
COMM MOVL C00224 BC00224 V=9.2
COMM MOVL C00225 BC00225 V=9.2
COMM MOVL C00226 BC00226 V=9.2
COMM SFTON P0402
COMM MOVL C00227 BC00227 V=9.2
COMM MOVL C00228 BC00228 V=9.2
COMM ARCOF
COMM MOVL C00229 BC00229 V=500.0
COMM SFTOF
COMM MOVJ C00230 BC00230 VJ=15.00
COMM 'W42B.1
COMM MOVJ C00231 BC00231 VJ=30.00
COMM MOVJ C00232 BC00232 VJ=30.00
COMM MOVJ C00233 BC00233 VJ=30.00
COMM MOVJ C00234 BC00234 VJ=30.00
COMM '**********************
COMM 'W42B.1
COMM '**********************
COMM MOVL C00235 BC00235 V=500.0
COMM SFTON P0399
COMM MOVL C00236 BC00236 V=66.7 PL=0
COMM MACRO1 MJ#(0) ARGF9
COMM ARCON
COMM SFTON P0415
COMM MOVL C00237 BC00237 V=9.2
COMM MOVL C00238 BC00238 V=9.2
COMM MOVL C00239 BC00239 V=9.2
COMM SFTON P0400
COMM MOVL C00240 BC00240 V=9.2
COMM MOVL C00241 BC00241 V=9.2
COMM ARCOF
COMM MOVL C00242 BC00242 V=500.0
COMM SFTOF
COMM MOVJ C00243 BC00243 VJ=15.00
COMM 'W42A.2
COMM MOVJ C00244 BC00244 VJ=20.00
COMM MOVJ C00245 BC00245 VJ=20.00
COMM MOVJ C00246 BC00246 VJ=20.00
COMM MOVJ C00247 BC00247 VJ=20.00
COMM MOVJ C00248 BC00248 VJ=20.00
COMM '**********************
COMM 'W42A.2
COMM '**********************
COMM MOVL C00249 BC00249 V=500.0
COMM SFTON P0402
COMM MOVL C00250 BC00250 V=66.7 PL=0
COMM SFTOF
COMM MACRO1 MJ#(0) ARGF9
COMM ARCON
COMM SFTON P0402
COMM MOVL C00251 BC00251 V=9.2
COMM ARCOF
COMM MOVL C00252 BC00252 V=166.7
COMM MOVJ C00253 BC00253 VJ=20.00
COMM MOVJ C00254 BC00254 VJ=20.00
COMM MOVL C00255 BC00255 V=166.7
COMM MOVL C00256 BC00256 V=166.7
COMM ARCON
COMM MOVL C00257 BC00257 V=10.8
COMM ARCOF
COMM MOVL C00258 BC00258 V=166.7
COMM MOVJ C00259 BC00259 VJ=10.00
COMM SFTOF
COMM MOVJ C00260 BC00260 VJ=20.00
COMM MOVJ C00261 BC00261 VJ=20.00
COMM MOVJ C00262 BC00262 VJ=20.00
COMM 'W42B.2
COMM MOVJ C00263 BC00263 VJ=20.00
COMM MOVJ C00264 BC00264 VJ=20.00
COMM MOVJ C00265 BC00265 VJ=20.00
COMM MOVJ C00266 BC00266 VJ=20.00
COMM MOVJ C00267 BC00267 VJ=20.00
COMM '**********************
COMM 'W42B.2
COMM '**********************
COMM MOVL C00268 BC00268 V=500.0
COMM SFTON P0400
COMM MOVL C00269 BC00269 V=166.7 PL=0
COMM SFTOF
COMM MACRO1 MJ#(0) ARGF9
COMM ARCON
COMM SFTON P0400
COMM MOVL C00270 BC00270 V=9.2
COMM ARCOF
COMM SFTOF
COMM MOVL C00271 BC00271 V=166.7
COMM MOVL C00272 BC00272 V=166.7
COMM MOVJ C00273 BC00273 VJ=10.00
COMM SFTON P0400
COMM MOVL C00274 BC00274 V=166.7
COMM ARCON
COMM MOVL C00275 BC00275 V=10.8
COMM ARCOF
COMM MOVL C00276 BC00276 V=166.7
COMM MOVL C00277 BC00277 V=500.0
COMM SFTOF
COMM MOVJ C00278 BC00278 VJ=20.00
COMM MOVJ C00279 BC00279 VJ=20.00
COMM 'W42A.3
COMM MOVJ C00280 BC00280 VJ=10.00
COMM MOVJ C00281 BC00281 VJ=20.00
COMM MOVJ C00282 BC00282 VJ=20.00
COMM MOVJ C00283 BC00283 VJ=20.00
COMM '**********************
COMM 'W42A.3
COMM '**********************
COMM MOVL C00284 BC00284 V=500.0
COMM SFTON P0402
COMM MOVL C00285 BC00285 V=166.7 PL=0
COMM MACRO1 MJ#(0) ARGF9
COMM ARCON
COMM MOVL C00286 BC00286 V=9.2
COMM ARCOF
COMM MOVL C00287 BC00287 V=500.0
COMM SFTOF
COMM '**********************
COMM 'W42B.3
COMM '**********************
COMM MOVL C00288 BC00288 V=500.0
COMM SFTON P0400
COMM MOVL C00289 BC00289 V=66.7 PL=0
COMM ARCON
COMM MOVL C00290 BC00290 V=9.2
COMM ARCOF
COMM MOVL C00291 BC00291 V=500.0
COMM SFTOF
COMM MOVJ C00292 BC00292 VJ=10.00
COMM '**********************
COMM 'GORA L
COMM '**********************
COMM MOVL C00293 BC00293 V=500.0
COMM SFTON P0401
COMM MOVL C00294 BC00294 V=66.7 PL=0
COMM MACRO1 MJ#(0) ARGF9
COMM ARCON
COMM MOVL C00295 BC00295 V=11.7
COMM SFTON P0406
COMM MOVL C00296 BC00296 V=11.7
COMM MOVL C00297 BC00297 V=11.7
COMM MOVL C00298 BC00298 V=11.7
COMM ARCOF
COMM MOVL C00299 BC00299 V=500.0
COMM SFTOF
COMM '**********************
COMM 'GORA P
COMM '**********************
COMM MOVL C00300 BC00300 V=166.7
COMM SFTON P0401
COMM MOVL C00301 BC00301 V=166.7 PL=0
COMM ARCON
COMM MOVL C00302 BC00302 V=11.7
COMM SFTON P0405
COMM MOVL C00303 BC00303 V=11.7
COMM MOVL C00304 BC00304 V=11.7
COMM MOVL C00305 BC00305 V=11.7
COMM ARCOF
COMM MOVL C00306 BC00306 V=500.0
COMM SFTOF
COMM MOVJ C00307 BC00307 VJ=10.00
COMM MOVJ C00308 BC00308 VJ=30.00
COMM MOVJ C00309 BC00309 VJ=30.00
COMM 'KONIEC SPAWANIA FRONTU
COMM '**********************
COMM 'W44
COMM '**********************
MOVJ C00310 BC00310 VJ=30.00
MOVJ C00311 BC00311 VJ=25.00
MOVJ C00312 BC00312 VJ=30.00
MOVJ C00313 BC00313 VJ=30.00
MOVL C00314 BC00314 V=500.0
SFTON P0108
MOVL C00315 BC00315 V=166.7 PL=0
SFTOF
MACRO1 MJ#(0) ARGF24
ARCON
SFTON P0107
MOVL C00316 BC00316 V=10.8
MOVL C00317 BC00317 V=10.8
ARCOF
SFTOF
MOVL C00318 BC00318 V=500.0
MOVL C00319 BC00319 V=500.0
MOVJ C00320 BC00320 VJ=30.00
'**********************
'W45
'**********************
MOVJ C00321 BC00321 VJ=30.00
MOVJ C00322 BC00322 VJ=20.00
MOVJ C00323 BC00323 VJ=10.00
MACRO1 MJ#(0) ARGF24
MOVL C00324 BC00324 V=500.0
SFTON P0102
MOVL C00325 BC00325 V=166.7 PL=0
SFTOF
ARCON
SFTON P0101
MOVL C00326 BC00326 V=12.5
ARCOF
SFTOF
MOVL C00327 BC00327 V=500.0
'**********************
'SPOINA_PODLOGA_BRAK_ROZP
'**********************
MOVL C00328 BC00328 V=500.0
MOVL C00329 BC00329 V=500.0
SFTON P0098
MOVL C00330 BC00330 V=166.7 PL=0
SFTOF
ARCON
SFTON P0097
MOVL C00331 BC00331 V=11.3
ARCOF
SFTOF
MOVL C00332 BC00332 V=166.7
'DODANE
MOVJ C00333 BC00333 VJ=10.00
MOVJ C00334 BC00334 VJ=10.00
'**********************
'W48
'**********************
MOVJ C00335 BC00335 VJ=15.00
MOVJ C00336 BC00336 VJ=25.00
MOVJ C00337 BC00337 VJ=15.00
SFTON P0104
MOVL C00338 BC00338 V=166.7 PL=0
SFTOF
ARCON
SFTON P0103
MOVL C00339 BC00339 V=10.5
ARCOF
SFTOF
MOVL C00340 BC00340 V=500.0
MOVJ C00341 BC00341 VJ=40.00
CALL JOB:FRONT_WELD_0ST-2_4840_V3
CALL JOB:MOVE_OUT_OF_TUNNEL
CALL JOB:CLEAN-R1
CALL JOB:MOVE_INTO_TUNNEL
MOVJ C00342 BC00342 VJ=30.00 PL=0
'------------------------
'------------------------
'PRAWA STRONA PROFIL GORA
'------------------------
'------------------------
MOVJ C00343 BC00343 VJ=20.00
'------------------------
'W51A L
'------------------------
SFTOF
MOVJ C00344 BC00344 VJ=10.00
MOVL C00345 BC00345 V=66.7 PL=0
REFP 3 C00346 BC00346
CALL JOB:SEARCH-R1
SET P0299 P0006
SFTON P0299
MOVL C00347 BC00347 V=66.7 PL=0
REFP 3 C00348 BC00348
CALL JOB:SEARCH-R1
SET P0299 P0006
SFTON P0299
MOVL C00349 BC00349 V=83.3
MOVL C00350 BC00350 V=166.7 PL=0
REFP 3 C00351 BC00351
CALL JOB:SEARCH-R1
SET P0299 P0006
SFTON P0299
MOVL C00352 BC00352 V=133.3 PL=0
SFTOF
'------------------------
'W51A P
'------------------------
SFTOF
MOVL C00353 BC00353 V=250.0
'------------------------
'W54A L
'------------------------
SFTOF
MOVJ C00354 BC00354 VJ=30.00
MOVL C00355 BC00355 V=133.3 PL=0
REFP 3 C00356 BC00356
CALL JOB:SEARCH-R1
SET P0301 P0006
SFTON P0301
MOVL C00357 BC00357 V=66.7 PL=0
REFP 3 C00358 BC00358
CALL JOB:SEARCH-R1
SET P0301 P0006
SFTON P0301
MOVL C00359 BC00359 V=66.7 PL=0
SFTOF
'------------------------
'W54A P
'------------------------
SFTOF
MOVJ C00360 BC00360 VJ=30.00
MOVL C00361 BC00361 V=133.3 PL=0
REFP 3 C00362 BC00362
CALL JOB:SEARCH-R1
SET P0302 P0006
SFTON P0302
MOVL C00363 BC00363 V=66.7 PL=0
REFP 3 C00364 BC00364
CALL JOB:SEARCH-R1
SET P0302 P0006
SFTON P0302
MOVL C00365 BC00365 V=66.7 PL=0
SFTOF
'------------------------
'W50A L
'------------------------
SFTOF
MOVJ C00366 BC00366 VJ=30.00
MOVL C00367 BC00367 V=133.3 PL=0
REFP 3 C00368 BC00368
CALL JOB:SEARCH-R1
SET P0303 P0006
SFTON P0303
MOVL C00369 BC00369 V=66.7 PL=0
REFP 3 C00370 BC00370
CALL JOB:SEARCH-R1
SET P0303 P0006
SFTON P0303
MOVL C00371 BC00371 V=66.7 PL=0
SFTOF
'------------------------
'W50A P
'------------------------
SFTOF
MOVJ C00372 BC00372 VJ=30.00
MOVL C00373 BC00373 V=133.3 PL=0
REFP 3 C00374 BC00374
CALL JOB:SEARCH-R1
SET P0304 P0006
SFTON P0304
MOVL C00375 BC00375 V=66.7 PL=0
REFP 3 C00376 BC00376
CALL JOB:SEARCH-R1
SET P0304 P0006
SFTON P0304
MOVL C00377 BC00377 V=66.7 PL=0
SFTOF
'------------------------
'W53A L
'------------------------
SFTOF
MOVJ C00378 BC00378 VJ=30.00
MOVL C00379 BC00379 V=133.3 PL=0
REFP 3 C00380 BC00380
CALL JOB:SEARCH-R1
SET P0305 P0006
SFTON P0305
MOVL C00381 BC00381 V=66.7 PL=0
REFP 3 C00382 BC00382
CALL JOB:SEARCH-R1
SET P0305 P0006
SFTON P0305
MOVL C00383 BC00383 V=66.7 PL=0
SFTOF
'------------------------
'W53A P
'------------------------
SFTOF
MOVJ C00384 BC00384 VJ=30.00
MOVL C00385 BC00385 V=200.0
MOVL C00386 BC00386 V=66.7 PL=0
REFP 3 C00387 BC00387
CALL JOB:SEARCH-R1
SET P0306 P0006
SFTON P0306
MOVL C00388 BC00388 V=66.7 PL=0
REFP 3 C00389 BC00389
CALL JOB:SEARCH-R1
SET P0306 P0006
SFTON P0306
MOVL C00390 BC00390 V=66.7 PL=0
SFTOF
'------------------------
'W56A L
'------------------------
SFTOF
MOVJ C00391 BC00391 VJ=30.00
MOVL C00392 BC00392 V=133.3 PL=0
REFP 3 C00393 BC00393
CALL JOB:SEARCH-R1
SET P0307 P0006
SFTON P0307
MOVL C00394 BC00394 V=66.7 PL=0
REFP 3 C00395 BC00395
CALL JOB:SEARCH-R1
SET P0307 P0006
SFTON P0307
MOVL C00396 BC00396 V=66.7 PL=0
SFTOF
'------------------------
'W56A P
'------------------------
SFTOF
MOVJ C00397 BC00397 VJ=30.00
MOVL C00398 BC00398 V=133.3 PL=0
REFP 3 C00399 BC00399
CALL JOB:SEARCH-R1
SET P0308 P0006
SFTON P0308
MOVL C00400 BC00400 V=66.7 PL=0
REFP 3 C00401 BC00401
CALL JOB:SEARCH-R1
SET P0308 P0006
SFTON P0308
MOVL C00402 BC00402 V=66.7 PL=0
SFTOF
'------------------------
SFTOF
MOVJ C00403 BC00403 VJ=30.00
MOVL C00404 BC00404 V=250.0
MOVL C00405 BC00405 V=66.7 PL=0
REFP 3 C00406 BC00406
CALL JOB:SEARCH-R1
SET P0309 P0006
SFTON P0309
MOVL C00407 BC00407 V=66.7 PL=0
REFP 3 C00408 BC00408
CALL JOB:SEARCH-R1
SET P0309 P0006
SFTON P0309
MOVL C00409 BC00409 V=66.7 PL=0
SFTOF
'------------------------
SFTOF
MOVJ C00410 BC00410 VJ=5.00
MOVJ C00411 BC00411 VJ=20.00
MOVL C00412 BC00412 V=116.7 PL=0
REFP 3 C00413 BC00413
CALL JOB:SEARCH-R1
SET P0310 P0006
SFTON P0310
MOVL C00414 BC00414 V=66.7 PL=0
REFP 3 C00415 BC00415
CALL JOB:SEARCH-R1
SET P0310 P0006
SFTON P0310
MOVL C00416 BC00416 V=66.7 PL=0
SFTOF
'------------------------
'W55A L
'------------------------
SFTOF
MOVL C00417 BC00417 V=250.0
MOVJ C00418 BC00418 VJ=10.00
MOVL C00419 BC00419 V=66.7 PL=0
REFP 3 C00420 BC00420
CALL JOB:SEARCH-R1
SET P0311 P0006
SFTON P0311
MOVL C00421 BC00421 V=66.7 PL=0
REFP 3 C00422 BC00422
CALL JOB:SEARCH-R1
SET P0311 P0006
SFTON P0311
MOVL C00423 BC00423 V=66.7 PL=0
SFTOF
'------------------------
'W55A P
'------------------------
SFTOF
MOVL C00424 BC00424 V=250.0
MOVL C00425 BC00425 V=166.7
MOVL C00426 BC00426 V=66.7 PL=0
REFP 3 C00427 BC00427
CALL JOB:SEARCH-R1
SET P0312 P0006
SFTON P0312
MOVL C00428 BC00428 V=66.7 PL=0
REFP 3 C00429 BC00429
CALL JOB:SEARCH-R1
SET P0312 P0006
SFTON P0312
MOVL C00430 BC00430 V=66.7 PL=0
MOVL C00431 BC00431 V=166.7
SFTOF
MOVL C00432 BC00432 V=250.0
MOVJ C00433 BC00433 VJ=20.00
MOVJ C00434 BC00434 VJ=20.00
MOVJ C00435 BC00435 VJ=20.00
MOVJ C00436 BC00436 VJ=20.00
MOVJ C00437 BC00437 VJ=20.00
MOVJ C00438 BC00438 VJ=20.00
'------------------------
'LEWA STRONA PROFIL GORA
'------------------------
MOVJ C00439 BC00439 VJ=10.00
'------------------------
SFTOF
MOVJ C00440 BC00440 VJ=10.00
MOVL C00441 BC00441 V=66.7 PL=0
REFP 3 C00442 BC00442
CALL JOB:SEARCH-R1
SET P0349 P0006
SFTON P0349
MOVL C00443 BC00443 V=66.7 PL=0
REFP 3 C00444 BC00444
CALL JOB:SEARCH-R1
SET P0349 P0006
SFTON P0349
MOVL C00445 BC00445 V=66.7 PL=0
SFTOF
MOVJ C00446 BC00446 VJ=10.00
MOVJ C00447 BC00447 VJ=10.00
'------------------------
'W55B P
'------------------------
SFTOF
MOVL C00448 BC00448 V=66.7 PL=0
REFP 3 C00449 BC00449
CALL JOB:SEARCH-R1
SET P0350 P0006
SFTON P0350
MOVL C00450 BC00450 V=66.7 PL=0
REFP 3 C00451 BC00451
CALL JOB:SEARCH-R1
SET P0350 P0006
SFTON P0350
MOVL C00452 BC00452 V=66.7 PL=0
SFTOF
'------------------------
'W52B L
'------------------------
SFTOF
MOVJ C00453 BC00453 VJ=20.00
MOVJ C00454 BC00454 VJ=20.00
MOVL C00455 BC00455 V=150.0
MOVL C00456 BC00456 V=66.7 PL=0
REFP 3 C00457 BC00457
CALL JOB:SEARCH-R1
SET P0351 P0006
SFTON P0351
MOVL C00458 BC00458 V=66.7 PL=0
REFP 3 C00459 BC00459
CALL JOB:SEARCH-R1
SET P0351 P0006
SFTON P0351
MOVL C00460 BC00460 V=66.7 PL=0
SFTOF
'------------------------
'W52B P
'------------------------
SFTOF
MOVJ C00461 BC00461 VJ=30.00
MOVL C00462 BC00462 V=116.7 PL=0
REFP 3 C00463 BC00463
CALL JOB:SEARCH-R1
SET P0352 P0006
SFTON P0352
MOVL C00464 BC00464 V=66.7 PL=0
REFP 3 C00465 BC00465
CALL JOB:SEARCH-R1
SET P0352 P0006
SFTON P0352
MOVL C00466 BC00466 V=66.7 PL=0
SFTOF
'------------------------
'W56B L
'------------------------
SFTOF
MOVJ C00467 BC00467 VJ=30.00
MOVL C00468 BC00468 V=116.7 PL=0
REFP 3 C00469 BC00469
CALL JOB:SEARCH-R1
SET P0353 P0006
SFTON P0353
MOVL C00470 BC00470 V=66.7 PL=0
REFP 3 C00471 BC00471
CALL JOB:SEARCH-R1
SET P0353 P0006
SFTON P0353
MOVL C00472 BC00472 V=66.7 PL=0
SFTOF
'------------------------
'W56B P
'------------------------
SFTOF
MOVJ C00473 BC00473 VJ=30.00
MOVL C00474 BC00474 V=116.7 PL=0
REFP 3 C00475 BC00475
CALL JOB:SEARCH-R1
SET P0354 P0006
SFTON P0354
MOVL C00476 BC00476 V=66.7 PL=0
REFP 3 C00477 BC00477
CALL JOB:SEARCH-R1
SET P0354 P0006
SFTON P0354
MOVL C00478 BC00478 V=66.7 PL=0
SFTOF
'------------------------
'W53B L
'------------------------
SFTOF
MOVJ C00479 BC00479 VJ=30.00
MOVL C00480 BC00480 V=116.7 PL=0
REFP 3 C00481 BC00481
CALL JOB:SEARCH-R1
SET P0355 P0006
SFTON P0355
MOVL C00482 BC00482 V=66.7 PL=0
REFP 3 C00483 BC00483
CALL JOB:SEARCH-R1
SET P0355 P0006
SFTON P0355
MOVL C00484 BC00484 V=66.7 PL=0
SFTOF
'------------------------
'W53B P
'------------------------
SFTOF
MOVJ C00485 BC00485 VJ=30.00
MOVL C00486 BC00486 V=116.7 PL=0
REFP 3 C00487 BC00487
CALL JOB:SEARCH-R1
SET P0356 P0006
SFTON P0356
MOVL C00488 BC00488 V=66.7 PL=0
REFP 3 C00489 BC00489
CALL JOB:SEARCH-R1
SET P0356 P0006
SFTON P0356
MOVL C00490 BC00490 V=66.7 PL=0
SFTOF
'------------------------
'W50B L
'------------------------
SFTOF
MOVJ C00491 BC00491 VJ=30.00
MOVL C00492 BC00492 V=116.7 PL=0
REFP 3 C00493 BC00493
CALL JOB:SEARCH-R1
SET P0357 P0006
SFTON P0357
MOVL C00494 BC00494 V=66.7 PL=0
REFP 3 C00495 BC00495
CALL JOB:SEARCH-R1
SET P0357 P0006
SFTON P0357
MOVL C00496 BC00496 V=66.7 PL=0
SFTOF
'------------------------
'W50B P
'------------------------
SFTOF
MOVJ C00497 BC00497 VJ=30.00
MOVL C00498 BC00498 V=116.7 PL=0
REFP 3 C00499 BC00499
CALL JOB:SEARCH-R1
SET P0358 P0006
SFTON P0358
MOVL C00500 BC00500 V=66.7 PL=0
REFP 3 C00501 BC00501
CALL JOB:SEARCH-R1
SET P0358 P0006
SFTON P0358
MOVL C00502 BC00502 V=66.7 PL=0
SFTOF
'------------------------
'W54B L
'------------------------
SFTOF
MOVJ C00503 BC00503 VJ=30.00
MOVL C00504 BC00504 V=116.7 PL=0
REFP 3 C00505 BC00505
CALL JOB:SEARCH-R1
SET P0359 P0006
SFTON P0359
MOVL C00506 BC00506 V=66.7 PL=0
REFP 3 C00507 BC00507
CALL JOB:SEARCH-R1
SET P0359 P0006
SFTON P0359
MOVL C00508 BC00508 V=66.7 PL=0
SFTOF
'------------------------
'W54B P
'------------------------
SFTOF
MOVJ C00509 BC00509 VJ=30.00
MOVL C00510 BC00510 V=116.7 PL=0
REFP 3 C00511 BC00511
CALL JOB:SEARCH-R1
SET P0360 P0006
SFTON P0360
MOVL C00512 BC00512 V=66.7 PL=0
REFP 3 C00513 BC00513
CALL JOB:SEARCH-R1
SET P0360 P0006
SFTON P0360
MOVL C00514 BC00514 V=166.7 PL=0
SFTOF
'------------------------
'W51B L
'------------------------
'------------------------
SFTOF
MOVL C00515 BC00515 V=150.0
MOVL C00516 BC00516 V=66.7 PL=0
REFP 3 C00517 BC00517
CALL JOB:SEARCH-R1
SET P0361 P0006
SFTON P0361
MOVL C00518 BC00518 V=66.7 PL=0
REFP 3 C00519 BC00519
CALL JOB:SEARCH-R1
SET P0361 P0006
SFTON P0361
MOVL C00520 BC00520 V=83.3
MOVL C00521 BC00521 V=133.3 PL=0
REFP 3 C00522 BC00522
CALL JOB:SEARCH-R1
SET P0361 P0006
SFTON P0361
SFTOF
MOVL C00523 BC00523 V=83.3
MOVJ C00524 BC00524 VJ=20.00
MOVJ C00525 BC00525 VJ=30.00
MOVJ C00526 BC00526 VJ=10.00
MOVJ C00527 BC00527 VJ=40.00
'**********************
'**********************
'POCZATEK SPAWANIA BOKI
'**********************
'**********************
MOVJ C00528 BC00528 VJ=30.00
MOVJ C00529 BC00529 VJ=20.00
'**********************
'W50A
'**********************
MOVL C00530 BC00530 V=250.0
SFTON P0304
MOVL C00531 BC00531 V=83.3 PL=0
SFTOF
MACRO1 MJ#(0) ARGF10
ARCON
SFTON P0303
MOVL C00532 BC00532 V=10.8
ARCOF
SFTOF
MOVL C00533 BC00533 V=250.0
'W13B
MOVJ C00534 BC00534 VJ=20.00
MOVJ C00535 BC00535 VJ=40.00
MOVJ C00536 BC00536 VJ=20.00
MOVJ C00537 BC00537 VJ=20.00
MOVJ C00538 BC00538 VJ=20.00
'**********************
'W50B
'**********************
MOVL C00539 BC00539 V=250.0
SFTON P0357
MOVL C00540 BC00540 V=166.7 PL=0
SFTOF
MACRO1 MJ#(0) ARGF10
ARCON
SFTON P0358
MOVL C00541 BC00541 V=10.8
ARCOF
SFTOF
MOVL C00542 BC00542 V=250.0
MOVJ C00543 BC00543 VJ=20.00
MOVJ C00544 BC00544 VJ=20.00
MOVJ C00545 BC00545 VJ=20.00
MOVJ C00546 BC00546 VJ=20.00
'**********************
'W51A
'**********************
MOVL C00547 BC00547 V=416.7
SFTON P0299
MOVL C00548 BC00548 V=166.7 PL=0
SFTOF
MACRO1 MJ#(0) ARGF10
ARCON
SFTON P0299
MOVL C00549 BC00549 V=10.8
MOVL C00550 BC00550 V=10.8
ARCOF
MOVL C00551 BC00551 V=166.7
MOVL C00552 BC00552 V=133.3 PL=0
ARCON
MOVL C00553 BC00553 V=8.3
ARCOF
SFTOF
MOVL C00554 BC00554 V=200.0
MOVJ C00555 BC00555 VJ=30.00
MOVJ C00556 BC00556 VJ=30.00
MOVJ C00557 BC00557 VJ=30.00
MOVJ C00558 BC00558 VJ=30.00
MOVJ C00559 BC00559 VJ=30.00
'**********************
'W51B
'**********************
MOVL C00560 BC00560 V=416.7
MOVL C00561 BC00561 V=416.7
SFTON P0361
MOVL C00562 BC00562 V=166.7 PL=0
SFTOF
MACRO1 MJ#(0) ARGF10
ARCON
SFTON P0362
MOVL C00563 BC00563 V=10.8
MOVL C00564 BC00564 V=10.8
ARCOF
MOVL C00565 BC00565 V=166.7
MACRO1 MJ#(0) ARGF9
MOVL C00566 BC00566 V=166.7 PL=0
ARCON
MOVL C00567 BC00567 V=8.3
ARCOF
SFTOF
MOVL C00568 BC00568 V=166.7
MOVL C00569 BC00569 V=250.0
MOVJ C00570 BC00570 VJ=30.00
MOVJ C00571 BC00571 VJ=30.00
MOVJ C00572 BC00572 VJ=30.00
MOVJ C00573 BC00573 VJ=40.00
MOVJ C00574 BC00574 VJ=40.00
MOVJ C00575 BC00575 VJ=20.00
MOVJ C00576 BC00576 VJ=20.00
MOVJ C00577 BC00577 VJ=20.00
MOVJ C00578 BC00578 VJ=20.00
MOVJ C00579 BC00579 VJ=20.00
'**********************
'W52A
'**********************
SFTON P0310
MOVL C00580 BC00580 V=250.0
MOVL C00581 BC00581 V=83.3 PL=0
SFTOF
MACRO1 MJ#(0) ARGF10
ARCON
SFTON P0309
MOVL C00582 BC00582 V=10.8
ARCOF
SFTOF
MOVL C00583 BC00583 V=333.3
MOVJ C00584 BC00584 VJ=30.00
MOVJ C00585 BC00585 VJ=30.00
MOVJ C00586 BC00586 VJ=30.00
MOVJ C00587 BC00587 VJ=30.00
MOVJ C00588 BC00588 VJ=30.00
MOVJ C00589 BC00589 VJ=20.00
MOVJ C00590 BC00590 VJ=20.00
MOVJ C00591 BC00591 VJ=20.00
'**********************
'52B
'**********************
MOVL C00592 BC00592 V=250.0
SFTON P0351
MOVL C00593 BC00593 V=83.3 PL=0
SFTOF
MACRO1 MJ#(0) ARGF10
ARCON
SFTON P0352
MOVL C00594 BC00594 V=10.8
ARCOF
MOVL C00595 BC00595 V=333.3
SFTOF
MOVJ C00596 BC00596 VJ=20.00
MOVJ C00597 BC00597 VJ=30.00
MOVJ C00598 BC00598 VJ=30.00
'**********************
'W53A
'**********************
MOVJ C00599 BC00599 VJ=30.00
MOVJ C00600 BC00600 VJ=30.00
MOVJ C00601 BC00601 VJ=10.00
'**********************
'W53A
'**********************
SFTON P0306
MOVL C00602 BC00602 V=250.0
MOVL C00603 BC00603 V=83.3 PL=0
SFTOF
MACRO1 MJ#(0) ARGF10
ARCON
SFTON P0305
MOVL C00604 BC00604 V=10.8
ARCOF
SFTOF
MOVL C00605 BC00605 V=250.0
MOVJ C00606 BC00606 VJ=30.00
MOVJ C00607 BC00607 VJ=30.00
MOVJ C00608 BC00608 VJ=30.00
MOVJ C00609 BC00609 VJ=30.00
MOVJ C00610 BC00610 VJ=30.00
MOVJ C00611 BC00611 VJ=30.00
MOVL C00612 BC00612 V=250.0
'**********************
'W53B
'**********************
SFTON P0355
MOVL C00613 BC00613 V=250.0
MOVL C00614 BC00614 V=83.3 PL=0
SFTOF
MACRO1 MJ#(0) ARGF10
ARCON
SFTON P0356
MOVL C00615 BC00615 V=10.8
ARCOF
SFTOF
MOVL C00616 BC00616 V=333.3
MOVJ C00617 BC00617 VJ=30.00
MOVJ C00618 BC00618 VJ=30.00
MOVJ C00619 BC00619 VJ=30.00
MOVJ C00620 BC00620 VJ=30.00
'**********************
'W54A
'**********************
SFTON P0302
MOVL C00621 BC00621 V=250.0
MOVL C00622 BC00622 V=83.3 PL=0
SFTOF
MACRO1 MJ#(0) ARGF10
ARCON
SFTON P0301
MOVL C00623 BC00623 V=10.8
ARCOF
SFTOF
MOVL C00624 BC00624 V=333.3
MOVJ C00625 BC00625 VJ=20.00
MOVJ C00626 BC00626 VJ=30.00
MOVJ C00627 BC00627 VJ=30.00
MOVJ C00628 BC00628 VJ=30.00
MOVJ C00629 BC00629 VJ=30.00
'**********************
'W54B
'**********************
SFTON P0359
MOVL C00630 BC00630 V=250.0
MOVL C00631 BC00631 V=83.3 PL=0
SFTOF
MACRO1 MJ#(0) ARGF10
ARCON
SFTON P0360
MOVL C00632 BC00632 V=10.8
ARCOF
MOVL C00633 BC00633 V=333.3
SFTOF
MOVJ C00634 BC00634 VJ=30.00
MOVJ C00635 BC00635 VJ=30.00
MOVJ C00636 BC00636 VJ=30.00
MOVJ C00637 BC00637 VJ=40.00
MOVJ C00638 BC00638 VJ=40.00
MOVJ C00639 BC00639 VJ=10.00
MOVJ C00640 BC00640 VJ=10.00
MOVJ C00641 BC00641 VJ=10.00
MOVJ C00642 BC00642 VJ=15.00
MOVJ C00643 BC00643 VJ=15.00
MOVJ C00644 BC00644 VJ=15.00
MOVJ C00645 BC00645 VJ=15.00
'**********************
'W55A
'**********************
SFTON P0311
MOVL C00646 BC00646 V=166.7 PL=0
SFTOF
MACRO1 MJ#(0) ARGF10
ARCON
SFTON P0312
MOVL C00647 BC00647 V=10.8
MOVL C00648 BC00648 V=10.8
ARCOF
SFTOF
MOVL C00649 BC00649 V=150.0
MOVJ C00650 BC00650 VJ=10.00
MOVJ C00651 BC00651 VJ=10.00
MOVJ C00652 BC00652 VJ=10.00
MOVJ C00653 BC00653 VJ=10.00
MOVJ C00654 BC00654 VJ=10.00
MOVJ C00655 BC00655 VJ=10.00
MOVJ C00656 BC00656 VJ=30.00
MOVJ C00657 BC00657 VJ=30.00
MOVJ C00658 BC00658 VJ=20.00
MOVJ C00659 BC00659 VJ=30.00
MOVJ C00660 BC00660 VJ=20.00
MOVJ C00661 BC00661 VJ=20.00
MOVJ C00662 BC00662 VJ=30.00
MOVJ C00663 BC00663 VJ=20.00
MOVJ C00664 BC00664 VJ=20.00
'**********************
'W55B
'**********************
SFTON P0350
MOVL C00665 BC00665 V=333.3
MOVL C00666 BC00666 V=166.7 PL=0
SFTOF
MACRO1 MJ#(0) ARGF10
ARCON
SFTON P0349
MOVL C00667 BC00667 V=10.8
MOVL C00668 BC00668 V=10.8
ARCOF
SFTOF
MOVL C00669 BC00669 V=66.7
MOVJ C00670 BC00670 VJ=10.00
MOVJ C00671 BC00671 VJ=20.00
MOVJ C00672 BC00672 VJ=20.00
MOVJ C00673 BC00673 VJ=20.00
MOVJ C00674 BC00674 VJ=30.00
MOVJ C00675 BC00675 VJ=50.00
MOVJ C00676 BC00676 VJ=50.00
MOVJ C00677 BC00677 VJ=40.00
MOVJ C00678 BC00678 VJ=20.00
'**********************
'W56A
'**********************
SFTON P0308
MOVL C00679 BC00679 V=333.3
MOVL C00680 BC00680 V=166.7 PL=0
SFTOF
MACRO1 MJ#(0) ARGF10
ARCON
SFTON P0307
MOVL C00681 BC00681 V=10.8
ARCOF
SFTOF
MOVL C00682 BC00682 V=333.3
MOVJ C00683 BC00683 VJ=20.00
MOVJ C00684 BC00684 VJ=30.00
MOVJ C00685 BC00685 VJ=30.00
MOVJ C00686 BC00686 VJ=30.00
'**********************
'W56B
'**********************
SFTON P0353
MOVL C00687 BC00687 V=250.0
MOVL C00688 BC00688 V=166.7 PL=0
SFTOF
MACRO1 MJ#(0) ARGF10
ARCON
SFTON P0354
MOVL C00689 BC00689 V=10.8
ARCOF
SFTOF
MOVL C00690 BC00690 V=333.3
MOVJ C00691 BC00691 VJ=30.00
MOVJ C00692 BC00692 VJ=30.00
MOVJ C00693 BC00693 VJ=30.00
CALL JOB:MOVE_OUT_OF_TUNNEL
CALL JOB:R1-HOME
END
